LIN {X 0,Y 452.05,Z 502.016,A -85,B 0,C 180,E1 -8755.313,E2 -8755.313} C_VEL
LIN {X 0,Y 450.081,Z 492.867,A -85,B 0,C 180,E1 -8757.12,E2 -8757.12} C_VEL
LIN {X 0,Y 447.199,Z 482.476,A -85,B 0,C 180,E1 -8759.407,E2 -8759.407} C_VEL
LIN {X 0,Y 446.433,Z 480.006,A -85,B 0,C 180,E1 -8760.021,E2 -8760.021} C_VEL
LIN {X 0,Y 446.447,Z 480.002,A -85,B 0,C 180,E1 -8763.454,E2 -8763.454} C_VEL
LIN {X 0,Y 446.404,Z 480.006,A -85,B 0,C 180,E1 -8766.745,E2 -8766.745} C_VEL
LIN {X 0,Y 446.471,Z 479.998,A -85,B 0,C 180,E1 -8769.527,E2 -8769.527} C_VEL
LIN {X 0,Y 446.435,Z 480,A -85,B 0,C 180,E1 -8772.604,E2 -8772.604} C_VEL
LIN {X 0,Y 446.457,Z 480,A -85,B 0,C 180,E1 -8775.103,E2 -8775.103} C_VEL
LIN {X 0,Y 446.431,Z 480.003,A -85,B 0,C 180,E1 -8778.609,E2 -8778.609} C_VEL
LIN {X 0,Y 446.459,Z 480,A -85,B 0,C 180,E1 -8780.974,E2 -8780.974} C_VEL
LIN {X 0,Y 446.423,Z 480.004,A -85,B 0,C 180,E1 -8784.374,E2 -8784.374} C_VEL
LIN {X 0,Y 446.426,Z 480.003,A -85,B 0,C 180,E1 -8787.639,E2 -8787.639} C_VEL
LIN {X 0,Y 446.453,Z 480.14,A -85,B 0,C 180,E1 -8790.791,E2 -8790.791} C_VEL
LIN {X 0,Y 449.137,Z 489.685,A -85,B 0,C 180,E1 -8793.117,E2 -8793.117} C_VEL
LIN {X 0,Y 451.239,Z 500.063,A -85,B 0,C 180,E1 -8795.378,E2 -8795.378} C_VEL
LIN {X 0,Y 451.318,Z 502.583,A -85,B 0,C 180,E1 -8795.872,E2 -8795.872} C_VEL
LIN {X 0,Y 449.674,Z 522.318,A -85,B 0,C 180,E1 -8799.459,E2 -8799.459} C_VEL
LIN {X 0,Y 448.638,Z 537.985,A -85,B 0,C 180,E1 -8802.214,E2 -8802.214} C_VEL
LIN {X 0,Y 448.559,Z 540.298,A -85,B 0,C 180,E1 -8802.575,E2 -8802.575} C_VEL
LIN {X 0,Y 451.577,Z 556.911,A -85,B 0,C 180,E1 -8803.122,E2 -8803.122} C_VEL
LIN {X 0,Y 452.097,Z 561.761,A -85,B 0,C 180,E1 -8803.261,E2 -8803.261} C_VEL
LIN {X 0,Y 450.024,Z 654.195,A -85,B 0,C 180,E1 -8805.183,E2 -8805.183} C_VEL
LIN {X 0,Y 449.587,Z 668.155,A -85,B 0,C 180,E1 -8805.66,E2 -8805.66} C_VEL
LIN {X 0,Y 449.12,Z 681.597,A -85,B 0,C 180,E1 -8806.333,E2 -8806.333} C_VEL
LIN {X 0,Y 448.59,Z 693.288,A -85,B 0,C 180,E1 -8807.1,E2 -8807.1} C_VEL
LIN {X 0,Y 447.989,Z 704.247,A -85,B 0,C 180,E1 -8808.003,E2 -8808.003} C_VEL
LIN {X 0,Y 447.339,Z 715.188,A -85,B 0,C 180,E1 -8809.133,E2 -8809.133} C_VEL
LIN {X 0,Y 446.903,Z 724.107,A -85,B 0,C 180,E1 -8810.267,E2 -8810.267} C_VEL
LIN {X 0,Y 446.363,Z 732.831,A -85,B 0,C 180,E1 -8811.626,E2 -8811.626} C_VEL
LIN {X 0,Y 446.034,Z 740.156,A -85,B 0,C 180,E1 -8813.06,E2 -8813.06} C_VEL
LIN {X 0,Y 445.863,Z 744.583,A -85,B 0,C 180,E1 -8814.119,E2 -8814.119} C_VEL
LIN {X 0,Y 445.641,Z 749.141,A -85,B 0,C 180,E1 -8815.477,E2 -8815.477} C_VEL
LIN {X 0,Y 445.638,Z 751.534,A -85,B 0,C 180,E1 -8816.383,E2 -8816.383} C_VEL
LIN {X 0,Y 445.507,Z 753.496,A -85,B 0,C 180,E1 -8817.287,E2 -8817.287} C_VEL
LIN {X 0,Y 445.412,Z 755.01,A -85,B 0,C 180,E1 -8818.192,E2 -8818.192} C_VEL
LIN {X 0,Y 445.37,Z 756.058,A -85,B 0,C 180,E1 -8819.096,E2 -8819.096} C_VEL
LIN {X 0,Y 445.343,Z 756.704,A -85,B 0,C 180,E1 -8820,E2 -8820} C_VEL
LIN {X 0,Y 445.341,Z 756.949,A -85,B 0,C 180,E1 -8820.904,E2 -8820.904} C_VEL
LIN {X 0,Y 445.379,Z 756.765,A -85,B 0,C 180,E1 -8821.809,E2 -8821.809} C_VEL
LIN {X 0,Y 445.453,Z 756.141,A -85,B 0,C 180,E1 -8822.713,E2 -8822.713} C_VEL
LIN {X 0,Y 445.442,Z 755.119,A -85,B 0,C 180,E1 -8823.618,E2 -8823.618} C_VEL
LIN {X 0,Y 445.439,Z 753.686,A -85,B 0,C 180,E1 -8824.525,E2 -8824.525} C_VEL
LIN {X 0,Y 445.583,Z 750.669,A -85,B 0,C 180,E1 -8825.884,E2 -8825.884} C_VEL
LIN {X 0,Y 445.669,Z 746.583,A -85,B 0,C 180,E1 -8827.248,E2 -8827.248} C_VEL
LIN {X 0,Y 445.945,Z 740.281,A -85,B 0,C 180,E1 -8828.839,E2 -8828.839} C_VEL
LIN {X 0,Y 446.236,Z 733.389,A -85,B 0,C 180,E1 -8830.206,E2 -8830.206} C_VEL
LIN {X 0,Y 446.731,Z 724.835,A -85,B 0,C 180,E1 -8831.571,E2 -8831.571} C_VEL
LIN {X 0,Y 447.063,Z 716.018,A -85,B 0,C 180,E1 -8832.714,E2 -8832.714} C_VEL
LIN {X 0,Y 447.647,Z 705.182,A -85,B 0,C 180,E1 -8833.852,E2 -8833.852} C_VEL
LIN {X 0,Y 448.271,Z 694.465,A -85,B 0,C 180,E1 -8834.76,E2 -8834.76} C_VEL
LIN {X 0,Y 448.76,Z 682.612,A -85,B 0,C 180,E1 -8835.557,E2 -8835.557} C_VEL
LIN {X 0,Y 449.237,Z 669.19,A -85,B 0,C 180,E1 -8836.239,E2 -8836.239} C_VEL
LIN {X 0,Y 449.601,Z 656.633,A -85,B 0,C 180,E1 -8836.692,E2 -8836.692} C_VEL
LIN {X 0,Y 449.911,Z 641.204,A -85,B 0,C 180,E1 -8837.031,E2 -8837.031} C_VEL
LIN {X 0,Y 451.097,Z 559.466,A -85,B 0,C 180,E1 -8838.551,E2 -8838.551} C_VEL
LIN {X 0,Y 448.101,Z 540.66,A -85,B 0,C 180,E1 -8839.052,E2 -8839.052} C_VEL
LIN {X 0,Y 449.102,Z 521.658,A -85,B 0,C 180,E1 -8842.27,E2 -8842.27} C_VEL
LIN {X 0,Y 450.259,Z 502.009,A -85,B 0,C 180,E1 -8845.642,E2 -8845.642} C_VEL
LIN {X 0,Y 450.32,Z 497.645,A -85,B 0,C 180,E1 -8846.41,E2 -8846.41} C_VEL
LIN {X 0,Y 447.487,Z 484.497,A -85,B 0,C 180,E1 -8848.933,E2 -8848.933} C_VEL
LIN {X 0,Y 446.441,Z 480.002,A -85,B 0,C 180,E1 -8849.823,E2 -8849.823} C_VEL
LIN {X 0,Y 446.451,Z 480.001,A -85,B 0,C 180,E1 -8853.433,E2 -8853.433} C_VEL
LIN {X 0,Y 446.411,Z 479.999,A -85,B 0,C 180,E1 -8856.744,E2 -8856.744} C_VEL
LIN {X 0,Y 446.481,Z 479.997,A -85,B 0,C 180,E1 -8859.528,E2 -8859.528} C_VEL
LIN {X 0,Y 446.431,Z 479.996,A -85,B 0,C 180,E1 -8862.604,E2 -8862.604} C_VEL
LIN {X 0,Y 446.454,Z 479.995,A -85,B 0,C 180,E1 -8865.103,E2 -8865.103} C_VEL
LIN {X 0,Y 446.43,Z 479.996,A -85,B 0,C 180,E1 -8868.609,E2 -8868.609} C_VEL
LIN {X 0,Y 446.44,Z 479.996,A -85,B 0,C 180,E1 -8870.972,E2 -8870.972} C_VEL
LIN {X 0,Y 446.421,Z 479.997,A -85,B 0,C 180,E1 -8874.374,E2 -8874.374} C_VEL
LIN {X 0,Y 446.424,Z 480.004,A -85,B 0,C 180,E1 -8877.638,E2 -8877.638} C_VEL
LIN {X 0,Y 446.45,Z 479.994,A -85,B 0,C 180,E1 -8880.791,E2 -8880.791} C_VEL
LIN {X 0,Y 446.461,Z 479.994,A -85,B 0,C 180,E1 -8884.111,E2 -8884.111} C_VEL
LIN {X 0,Y 446.43,Z 479.997,A -85,B 0,C 180,E1 -8886.823,E2 -8886.823} C_VEL
LIN {X 0,Y 446.433,Z 479.998,A -85,B 0,C 180,E1 -8888.036,E2 -8888.036} C_VEL
LIN {X 0,Y 445.804,Z 480.076,A -85,B 0,C 180,E1 -8888.79,E2 -8888.79} C_VEL
LIN {X 0,Y 442.953,Z 480.431,A -85,B 0,C 180,E1 -8890.015,E2 -8890.015} C_VEL
LIN {X 0,Y 440.525,Z 480.734,A -85,B 0,C 180,E1 -8891.003,E2 -8891.003} C_VEL
LIN {X 0,Y 439.495,Z 480.864,A -85,B 0,C 180,E1 -8891.767,E2 -8891.767} C_VEL
LIN {X 0,Y 439.42,Z 480.87,A -85,B 0,C 180,E1 -8892.025,E2 -8892.025} C_VEL
LIN {X 0,Y 439.451,Z 480.869,A -85,B 0,C 180,E1 -8895.174,E2 -8895.174} C_VEL
LIN {X 0,Y 439.486,Z 480.863,A -85,B 0,C 180,E1 -8898.001,E2 -8898.001} C_VEL
LIN {X 0,Y 439.55,Z 480.858,A -85,B 0,C 180,E1 -8901.726,E2 -8901.726} C_VEL
LIN {X 0,Y 439.623,Z 480.844,A -85,B 0,C 180,E1 -8904.496,E2 -8904.496} C_VEL
LIN {X 0,Y 439.637,Z 480.843,A -85,B 0,C 180,E1 -8908.168,E2 -8908.168} C_VEL
LIN {X 0,Y 439.766,Z 480.828,A -85,B 0,C 180,E1 -8910,E2 -8910} C_VEL
LIN {X 0,Y 439.658,Z 480.84,A -85,B 0,C 180,E1 -8912.749,E2 -8912.749} C_VEL
LIN {X 0,Y 439.615,Z 480.845,A -85,B 0,C 180,E1 -8916.425,E2 -8916.425} C_VEL
LIN {X 0,Y 439.501,Z 480.864,A -85,B 0,C 180,E1 -8919.202,E2 -8919.202} C_VEL
LIN {X 0,Y 439.467,Z 480.866,A -85,B 0,C 180,E1 -8922.938,E2 -8922.938} C_VEL
LIN {X 0,Y 439.449,Z 480.866,A -85,B 0,C 180,E1 -8926.349,E2 -8926.349} C_VEL
LIN {X 0,Y 439.404,Z 480.876,A -85,B 0,C 180,E1 -8929.626,E2 -8929.626} C_VEL
LIN {X 0,Y 439.367,Z 480.876,A -85,B 0,C 180,E1 -8932.575,E2 -8932.575} C_VEL
LIN {X 0,Y 439.407,Z 480.876,A -85,B 0,C 180,E1 -8935.585,E2 -8935.585} C_VEL
LIN {X 0,Y 439.419,Z 480.87,A -85,B 0,C 180,E1 -8938.673,E2 -8938.673} C_VEL
LIN {X 0,Y 439.372,Z 480.876,A -85,B 0,C 180,E1 -8942.031,E2 -8942.031} C_VEL
LIN {X 0,Y 439.396,Z 480.881,A -85,B 0,C 180,E1 -8945.34,E2 -8945.34} C_VEL
LIN {X 0,Y 439.386,Z 480.874,A -85,B 0,C 180,E1 -8948.595,E2 -8948.595} C_VEL
LIN {X 0,Y 439.391,Z 480.88,A -85,B 0,C 180,E1 -8951.257,E2 -8951.257} C_VEL
LIN {X 0,Y 439.407,Z 480.872,A -85,B 0,C 180,E1 -8954.729,E2 -8954.729} C_VEL
LIN {X 0,Y 439.397,Z 480.874,A -85,B 0,C 180,E1 -8957.796,E2 -8957.796} C_VEL
LIN {X 0,Y 439.427,Z 480.868,A -85,B 0,C 180,E1 -8960.227,E2 -8960.227} C_VEL
LIN {X 0,Y 439.376,Z 480.878,A -85,B 0,C 180,E1 -8963.713,E2 -8963.713} C_VEL
LIN {X 0,Y 439.375,Z 480.88,A -85,B 0,C 180,E1 -8967.054,E2 -8967.054} C_VEL
LIN {X 0,Y 439.385,Z 480.875,A -85,B 0,C 180,E1 -8970.274,E2 -8970.274} C_VEL
LIN {X 0,Y 439.435,Z 480.978,A -85,B 0,C 180,E1 -8971.598,E2 -8971.598} C_VEL
LIN {X 0,Y 442.64,Z 495.633,A -85,B 0,C 180,E1 -8974.111,E2 -8974.111} C_VEL
LIN {X 0,Y 443.148,Z 500.066,A -85,B 0,C 180,E1 -8974.835,E2 -8974.835} C_VEL
LIN {X 0,Y 442.278,Z 520.819,A -85,B 0,C 180,E1 -8978.073,E2 -8978.073} C_VEL
LIN {X 0,Y 441.486,Z 540.87,A -85,B 0,C 180,E1 -8981.194,E2 -8981.194} C_VEL
LIN {X 0,Y 441.286,Z 546.526,A -85,B 0,C 180,E1 -8982.072,E2 -8982.072} C_VEL
LIN {X 0,Y 443.899,Z 564.854,A -85,B 0,C 180,E1 -8982.535,E2 -8982.535} C_VEL
LIN {X 0,Y 442.597,Z 656.535,A -85,B 0,C 180,E1 -8984.251,E2 -8984.251} C_VEL
LIN {X 0,Y 442.194,Z 670.017,A -85,B 0,C 180,E1 -8984.679,E2 -8984.679} C_VEL
LIN {X 0,Y 441.715,Z 683.289,A -85,B 0,C 180,E1 -8985.311,E2 -8985.311} C_VEL
LIN {X 0,Y 441.247,Z 695.084,A -85,B 0,C 180,E1 -8986.06,E2 -8986.06} C_VEL
LIN {X 0,Y 440.748,Z 706.198,A -85,B 0,C 180,E1 -8986.968,E2 -8986.968} C_VEL
LIN {X 0,Y 440.215,Z 716.607,A -85,B 0,C 180,E1 -8988.022,E2 -8988.022} C_VEL
LIN {X 0,Y 439.718,Z 725.882,A -85,B 0,C 180,E1 -8989.176,E2 -8989.176} C_VEL
LIN {X 0,Y 439.212,Z 734.842,A -85,B 0,C 180,E1 -8990.56,E2 -8990.56} C_VEL
LIN {X 0,Y 438.87,Z 742.06,A -85,B 0,C 180,E1 -8991.945,E2 -8991.945} C_VEL
LIN {X 0,Y 438.645,Z 748.027,A -85,B 0,C 180,E1 -8993.4,E2 -8993.4} C_VEL
LIN {X 0,Y 438.471,Z 752.884,A -85,B 0,C 180,E1 -8994.942,E2 -8994.942} C_VEL
LIN {X 0,Y 438.383,Z 756.075,A -85,B 0,C 180,E1 -8996.323,E2 -8996.323} C_VEL
LIN {X 0,Y 438.389,Z 757.657,A -85,B 0,C 180,E1 -8997.243,E2 -8997.243} C_VEL
LIN {X 0,Y 438.301,Z 758.768,A -85,B 0,C 180,E1 -8998.162,E2 -8998.162} C_VEL
LIN {X 0,Y 438.255,Z 759.464,A -85,B 0,C 180,E1 -8999.081,E2 -8999.081} C_VEL
LIN {X 0,Y 438.253,Z 759.761,A -85,B 0,C 180,E1 -9000,E2 -9000} C_VEL
LIN {X 0,Y 438.255,Z 759.622,A -85,B 0,C 180,E1 -9000.919,E2 -9000.919} C_VEL
LIN {X 0,Y 438.3,Z 759.044,A -85,B 0,C 180,E1 -9001.838,E2 -9001.838} C_VEL
LIN {X 0,Y 438.391,Z 758.064,A -85,B 0,C 180,E1 -9002.757,E2 -9002.757} C_VEL
LIN {X 0,Y 438.404,Z 756.662,A -85,B 0,C 180,E1 -9003.677,E2 -9003.677} C_VEL
LIN {X 0,Y 438.471,Z 753.693,A -85,B 0,C 180,E1 -9005.058,E2 -9005.058} C_VEL
LIN {X 0,Y 438.728,Z 748.75,A -85,B 0,C 180,E1 -9006.693,E2 -9006.693} C_VEL
LIN {X 0,Y 438.971,Z 742.362,A -85,B 0,C 180,E1 -9008.285,E2 -9008.285} C_VEL
LIN {X 0,Y 439.365,Z 735.209,A -85,B 0,C 180,E1 -9009.669,E2 -9009.669} C_VEL
LIN {X 0,Y 439.835,Z 726.323,A -85,B 0,C 180,E1 -9011.055,E2 -9011.055} C_VEL
LIN {X 0,Y 440.485,Z 716.065,A -85,B 0,C 180,E1 -9012.322,E2 -9012.322} C_VEL
LIN {X 0,Y 441.026,Z 705.55,A -85,B 0,C 180,E1 -9013.371,E2 -9013.371} C_VEL
LIN {X 0,Y 441.563,Z 694.039,A -85,B 0,C 180,E1 -9014.282,E2 -9014.282} C_VEL
LIN {X 0,Y 442.067,Z 682.933,A -85,B 0,C 180,E1 -9014.972,E2 -9014.972} C_VEL
LIN {X 0,Y 442.533,Z 670.892,A -85,B 0,C 180,E1 -9015.545,E2 -9015.545} C_VEL
LIN {X 0,Y 442.905,Z 657.826,A -85,B 0,C 180,E1 -9015.975,E2 -9015.975} C_VEL
LIN {X 0,Y 444.641,Z 563.555,A -85,B 0,C 180,E1 -9017.869,E2 -9017.869} C_VEL
LIN {X 0,Y 441.922,Z 547.719,A -85,B 0,C 180,E1 -9018.368,E2 -9018.368} C_VEL
LIN {X 0,Y 442.726,Z 526.147,A -85,B 0,C 180,E1 -9021.659,E2 -9021.659} C_VEL
LIN {X 0,Y 443.633,Z 505.304,A -85,B 0,C 180,E1 -9024.823,E2 -9024.823} C_VEL
LIN {X 0,Y 443.662,Z 498.749,A -85,B 0,C 180,E1 -9025.825,E2 -9025.825} C_VEL
LIN {X 0,Y 441.267,Z 487.476,A -85,B 0,C 180,E1 -9027.744,E2 -9027.744} C_VEL
LIN {X 0,Y 439.446,Z 480.874,A -85,B 0,C 180,E1 -9028.933,E2 -9028.933} C_VEL
LIN {X 0,Y 439.373,Z 480.884,A -85,B 0,C 180,E1 -9032.03,E2 -9032.03} C_VEL
LIN {X 0,Y 439.397,Z 480.878,A -85,B 0,C 180,E1 -9035.34,E2 -9035.34} C_VEL
LIN {X 0,Y 439.385,Z 480.879,A -85,B 0,C 180,E1 -9038.595,E2 -9038.595} C_VEL
LIN {X 0,Y 439.39,Z 480.877,A -85,B 0,C 180,E1 -9041.257,E2 -9041.257} C_VEL
LIN {X 0,Y 439.404,Z 480.877,A -85,B 0,C 180,E1 -9044.729,E2 -9044.729} C_VEL
LIN {X 0,Y 439.4,Z 480.875,A -85,B 0,C 180,E1 -9047.796,E2 -9047.796} C_VEL
LIN {X 0,Y 439.439,Z 480.874,A -85,B 0,C 180,E1 -9050.228,E2 -9050.228} C_VEL
LIN {X 0,Y 439.379,Z 480.878,A -85,B 0,C 180,E1 -9053.713,E2 -9053.713} C_VEL
LIN {X 0,Y 439.377,Z 480.879,A -85,B 0,C 180,E1 -9057.054,E2 -9057.054} C_VEL
LIN {X 0,Y 439.438,Z 480.874,A -85,B 0,C 180,E1 -9060.804,E2 -9060.804} C_VEL
LIN {X 0,Y 439.474,Z 480.999,A -85,B 0,C 180,E1 -9061.233,E2 -9061.233} C_VEL
LIN {X 0,Y 443.439,Z 497.52,A -85,B 0,C 180,E1 -9064.149,E2 -9064.149} C_VEL
LIN {X 0,Y 444.397,Z 502.382,A -85,B 0,C 180,E1 -9064.973,E2 -9064.973} C_VEL
LIN {X 0,Y 442.89,Z 524.545,A -85,B 0,C 180,E1 -9068.35,E2 -9068.35} C_VEL
LIN {X 0,Y 442.849,Z 525.695,A -85,B 0,C 180,E1 -9068.485,E2 -9068.485} C_VEL
LIN {X 0,Y 445.968,Z 545.988,A -85,B 0,C 180,E1 -9069.007,E2 -9069.007} C_VEL
LIN {X 0,Y 444.046,Z 662.624,A -85,B 0,C 180,E1 -9071.127,E2 -9071.127} C_VEL
LIN {X 0,Y 443.555,Z 677.086,A -85,B 0,C 180,E1 -9071.575,E2 -9071.575} C_VEL
LIN {X 0,Y 443.021,Z 691.131,A -85,B 0,C 180,E1 -9072.204,E2 -9072.204} C_VEL
LIN {X 0,Y 442.484,Z 703.157,A -85,B 0,C 180,E1 -9072.912,E2 -9072.912} C_VEL
LIN {X 0,Y 441.698,Z 715.682,A -85,B 0,C 180,E1 -9073.832,E2 -9073.832} C_VEL
LIN {X 0,Y 441.014,Z 727.136,A -85,B 0,C 180,E1 -9074.873,E2 -9074.873} C_VEL
LIN {X 0,Y 440.246,Z 738.604,A -85,B 0,C 180,E1 -9076.145,E2 -9076.145} C_VEL
LIN {X 0,Y 439.747,Z 748.996,A -85,B 0,C 180,E1 -9077.566,E2 -9077.566} C_VEL
LIN {X 0,Y 439.237,Z 757.274,A -85,B 0,C 180,E1 -9078.93,E2 -9078.93} C_VEL
LIN {X 0,Y 438.83,Z 765.321,A -85,B 0,C 180,E1 -9080.552,E2 -9080.552} C_VEL
LIN {X 0,Y 438.529,Z 771.754,A -85,B 0,C 180,E1 -9082.171,E2 -9082.171} C_VEL
LIN {X 0,Y 438.442,Z 776.349,A -85,B 0,C 180,E1 -9083.631,E2 -9083.631} C_VEL
LIN {X 0,Y 438.321,Z 780.535,A -85,B 0,C 180,E1 -9085.402,E2 -9085.402} C_VEL
LIN {X 0,Y 438.337,Z 783.411,A -85,B 0,C 180,E1 -9087.243,E2 -9087.243} C_VEL
LIN {X 0,Y 438.252,Z 784.843,A -85,B 0,C 180,E1 -9089.081,E2 -9089.081} C_VEL
LIN {X 0,Y 438.252,Z 784.854,A -85,B 0,C 180,E1 -9090.919,E2 -9090.919} C_VEL
LIN {X 0,Y 438.337,Z 783.426,A -85,B 0,C 180,E1 -9092.757,E2 -9092.757} C_VEL
LIN {X 0,Y 438.321,Z 780.547,A -85,B 0,C 180,E1 -9094.598,E2 -9094.598} C_VEL
LIN {X 0,Y 438.447,Z 776.153,A -85,B 0,C 180,E1 -9096.443,E2 -9096.443} C_VEL
LIN {X 0,Y 438.525,Z 771.78,A -85,B 0,C 180,E1 -9097.83,E2 -9097.83} C_VEL
LIN {X 0,Y 438.818,Z 765.357,A -85,B 0,C 180,E1 -9099.449,E2 -9099.449} C_VEL
LIN {X 0,Y 439.232,Z 757.324,A -85,B 0,C 180,E1 -9101.07,E2 -9101.07} C_VEL
LIN {X 0,Y 439.779,Z 748.08,A -85,B 0,C 180,E1 -9102.587,E2 -9102.587} C_VEL
LIN {X 0,Y 440.295,Z 738.736,A -85,B 0,C 180,E1 -9103.853,E2 -9103.853} C_VEL
LIN {X 0,Y 440.979,Z 727.39,A -85,B 0,C 180,E1 -9105.128,E2 -9105.128} C_VEL
LIN {X 0,Y 441.687,Z 716.073,A -85,B 0,C 180,E1 -9106.168,E2 -9106.168} C_VEL
LIN {X 0,Y 442.483,Z 703.72,A -85,B 0,C 180,E1 -9107.088,E2 -9107.088} C_VEL
LIN {X 0,Y 443.135,Z 690.483,A -85,B 0,C 180,E1 -9107.87,E2 -9107.87} C_VEL
LIN {X 0,Y 443.743,Z 675.682,A -85,B 0,C 180,E1 -9108.527,E2 -9108.527} C_VEL
LIN {X 0,Y 444.265,Z 661.645,A -85,B 0,C 180,E1 -9108.953,E2 -9108.953} C_VEL
LIN {X 0,Y 446.318,Z 552.911,A -85,B 0,C 180,E1 -9111.032,E2 -9111.032} C_VEL
LIN {X 0,Y 446.402,Z 545.094,A -85,B 0,C 180,E1 -9111.194,E2 -9111.194} C_VEL
LIN {X 0,Y 444.191,Z 530.718,A -85,B 0,C 180,E1 -9111.634,E2 -9111.634} C_VEL
LIN {X 0,Y 443.391,Z 526.521,A -85,B 0,C 180,E1 -9111.793,E2 -9111.793} C_VEL
LIN {X 0,Y 445.31,Z 507.027,A -85,B 0,C 180,E1 -9114.972,E2 -9114.972} C_VEL
LIN {X 0,Y 445.319,Z 503.632,A -85,B 0,C 180,E1 -9115.58,E2 -9115.58} C_VEL
LIN {X 0,Y 443.118,Z 493.62,A -85,B 0,C 180,E1 -9117.64,E2 -9117.64} C_VEL
LIN {X 0,Y 439.987,Z 482.961,A -85,B 0,C 180,E1 -9120.132,E2 -9120.132} C_VEL
LIN {X 0,Y 439.362,Z 480.886,A -85,B 0,C 180,E1 -9120.712,E2 -9120.712} C_VEL
LIN {X 0,Y 439.389,Z 480.88,A -85,B 0,C 180,E1 -9124.044,E2 -9124.044} C_VEL
LIN {X 0,Y 439.35,Z 480.884,A -85,B 0,C 180,E1 -9126.887,E2 -9126.887} C_VEL
LIN {X 0,Y 439.409,Z 480.876,A -85,B 0,C 180,E1 -9129.85,E2 -9129.85} C_VEL
LIN {X 0,Y 439.388,Z 480.878,A -85,B 0,C 180,E1 -9132.628,E2 -9132.628} C_VEL
LIN {X 0,Y 439.405,Z 480.877,A -85,B 0,C 180,E1 -9135.271,E2 -9135.271} C_VEL
LIN {X 0,Y 439.391,Z 480.88,A -85,B 0,C 180,E1 -9138.743,E2 -9138.743} C_VEL
LIN {X 0,Y 439.379,Z 480.881,A -85,B 0,C 180,E1 -9141.607,E2 -9141.607} C_VEL
LIN {X 0,Y 439.402,Z 480.88,A -85,B 0,C 180,E1 -9144.844,E2 -9144.844} C_VEL
LIN {X 0,Y 439.377,Z 480.881,A -85,B 0,C 180,E1 -9148.14,E2 -9148.14} C_VEL
LIN {X 0,Y 439.401,Z 480.972,A -85,B 0,C 180,E1 -9150.137,E2 -9150.137} C_VEL
LIN {X 0,Y 442.403,Z 491.514,A -85,B 0,C 180,E1 -9152.825,E2 -9152.825} C_VEL
LIN {X 0,Y 444.372,Z 500.982,A -85,B 0,C 180,E1 -9154.972,E2 -9154.972} C_VEL
LIN {X 0,Y 444.725,Z 503.411,A -85,B 0,C 180,E1 -9155.491,E2 -9155.491} C_VEL
LIN {X 0,Y 442.962,Z 523.022,A -85,B 0,C 180,E1 -9159.134,E2 -9159.134} C_VEL
LIN {X 0,Y 441.785,Z 539.267,A -85,B 0,C 180,E1 -9162.052,E2 -9162.052} C_VEL
LIN {X 0,Y 441.805,Z 540.203,A -85,B 0,C 180,E1 -9162.169,E2 -9162.169} C_VEL
LIN {X 0,Y 444.963,Z 557.327,A -85,B 0,C 180,E1 -9162.771,E2 -9162.771} C_VEL
LIN {X 0,Y 445.523,Z 562.72,A -85,B 0,C 180,E1 -9162.932,E2 -9162.932} C_VEL
LIN {X 0,Y 443.28,Z 654.232,A -85,B 0,C 180,E1 -9164.894,E2 -9164.894} C_VEL
LIN {X 0,Y 442.83,Z 668.089,A -85,B 0,C 180,E1 -9165.38,E2 -9165.38} C_VEL
LIN {X 0,Y 442.356,Z 681.069,A -85,B 0,C 180,E1 -9166.037,E2 -9166.037} C_VEL
LIN {X 0,Y 441.706,Z 693.958,A -85,B 0,C 180,E1 -9166.895,E2 -9166.895} C_VEL
LIN {X 0,Y 441.074,Z 704.807,A -85,B 0,C 180,E1 -9167.812,E2 -9167.812} C_VEL
LIN {X 0,Y 440.396,Z 715.704,A -85,B 0,C 180,E1 -9168.96,E2 -9168.96} C_VEL
LIN {X 0,Y 439.932,Z 724.592,A -85,B 0,C 180,E1 -9170.111,E2 -9170.111} C_VEL
LIN {X 0,Y 439.355,Z 733.264,A -85,B 0,C 180,E1 -9171.491,E2 -9171.491} C_VEL
LIN {X 0,Y 438.987,Z 740.884,A -85,B 0,C 180,E1 -9173.026,E2 -9173.026} C_VEL
LIN {X 0,Y 438.83,Z 744.93,A -85,B 0,C 180,E1 -9174.025,E2 -9174.025} C_VEL
LIN {X 0,Y 438.557,Z 749.459,A -85,B 0,C 180,E1 -9175.404,E2 -9175.404} C_VEL
LIN {X 0,Y 438.582,Z 751.844,A -85,B 0,C 180,E1 -9176.325,E2 -9176.325} C_VEL
LIN {X 0,Y 438.438,Z 753.797,A -85,B 0,C 180,E1 -9177.244,E2 -9177.244} C_VEL
LIN {X 0,Y 438.332,Z 755.289,A -85,B 0,C 180,E1 -9178.162,E2 -9178.162} C_VEL
LIN {X 0,Y 438.282,Z 756.326,A -85,B 0,C 180,E1 -9179.081,E2 -9179.081} C_VEL
LIN {X 0,Y 438.254,Z 756.958,A -85,B 0,C 180,E1 -9180,E2 -9180} C_VEL
LIN {X 0,Y 438.255,Z 757.187,A -85,B 0,C 180,E1 -9180.919,E2 -9180.919} C_VEL
LIN {X 0,Y 438.3,Z 756.97,A -85,B 0,C 180,E1 -9181.838,E2 -9181.838} C_VEL
LIN {X 0,Y 438.38,Z 756.327,A -85,B 0,C 180,E1 -9182.757,E2 -9182.757} C_VEL
LIN {X 0,Y 438.344,Z 755.28,A -85,B 0,C 180,E1 -9183.677,E2 -9183.677} C_VEL
LIN {X 0,Y 438.365,Z 753.819,A -85,B 0,C 180,E1 -9184.598,E2 -9184.598} C_VEL
LIN {X 0,Y 438.487,Z 750.335,A -85,B 0,C 180,E1 -9186.136,E2 -9186.136} C_VEL
LIN {X 0,Y 438.681,Z 744.948,A -85,B 0,C 180,E1 -9187.827,E2 -9187.827} C_VEL
LIN {X 0,Y 438.937,Z 739.175,A -85,B 0,C 180,E1 -9189.213,E2 -9189.213} C_VEL
LIN {X 0,Y 439.254,Z 731.96,A -85,B 0,C 180,E1 -9190.603,E2 -9190.603} C_VEL
LIN {X 0,Y 439.824,Z 722.925,A -85,B 0,C 180,E1 -9191.989,E2 -9191.989} C_VEL
LIN {X 0,Y 440.223,Z 713.82,A -85,B 0,C 180,E1 -9193.132,E2 -9193.132} C_VEL
LIN {X 0,Y 440.811,Z 703.502,A -85,B 0,C 180,E1 -9194.189,E2 -9194.189} C_VEL
LIN {X 0,Y 441.458,Z 692.254,A -85,B 0,C 180,E1 -9195.111,E2 -9195.111} C_VEL
LIN {X 0,Y 441.966,Z 679.765,A -85,B 0,C 180,E1 -9195.921,E2 -9195.921} C_VEL
LIN {X 0,Y 442.355,Z 668.048,A -85,B 0,C 180,E1 -9196.499,E2 -9196.499} C_VEL
LIN {X 0,Y 442.822,Z 654.749,A -85,B 0,C 180,E1 -9196.955,E2 -9196.955} C_VEL
LIN {X 0,Y 443.146,Z 636.912,A -85,B 0,C 180,E1 -9197.329,E2 -9197.329} C_VEL
LIN {X 0,Y 444.371,Z 560.785,A -85,B 0,C 180,E1 -9198.784,E2 -9198.784} C_VEL
LIN {X 0,Y 441.168,Z 540.605,A -85,B 0,C 180,E1 -9199.333,E2 -9199.333} C_VEL
LIN {X 0,Y 442.387,Z 519.198,A -85,B 0,C 180,E1 -9203.011,E2 -9203.011} C_VEL
LIN {X 0,Y 443.532,Z 500.154,A -85,B 0,C 180,E1 -9206.339,E2 -9206.339} C_VEL
LIN {X 0,Y 441.231,Z 488.712,A -85,B 0,C 180,E1 -9208.545,E2 -9208.545} C_VEL
LIN {X 0,Y 439.403,Z 480.878,A -85,B 0,C 180,E1 -9210.134,E2 -9210.134} C_VEL
LIN {X 0,Y 439.399,Z 480.879,A -85,B 0,C 180,E1 -9213.724,E2 -9213.724} C_VEL
LIN {X 0,Y 439.359,Z 480.878,A -85,B 0,C 180,E1 -9216.888,E2 -9216.888} C_VEL
LIN {X 0,Y 439.415,Z 480.875,A -85,B 0,C 180,E1 -9219.851,E2 -9219.851} C_VEL
LIN {X 0,Y 439.384,Z 480.874,A -85,B 0,C 180,E1 -9222.627,E2 -9222.627} C_VEL
LIN {X 0,Y 439.402,Z 480.876,A -85,B 0,C 180,E1 -9225.27,E2 -9225.27} C_VEL
LIN {X 0,Y 439.39,Z 480.873,A -85,B 0,C 180,E1 -9228.743,E2 -9228.743} C_VEL
LIN {X 0,Y 439.374,Z 480.883,A -85,B 0,C 180,E1 -9231.608,E2 -9231.608} C_VEL
LIN {X 0,Y 439.401,Z 480.872,A -85,B 0,C 180,E1 -9234.844,E2 -9234.844} C_VEL
LIN {X 0,Y 439.375,Z 480.876,A -85,B 0,C 180,E1 -9238.139,E2 -9238.139} C_VEL
LIN {X 0,Y 439.434,Z 480.875,A -85,B 0,C 180,E1 -9241.598,E2 -9241.598} C_VEL
LIN {X 0,Y 439.407,Z 480.871,A -85,B 0,C 180,E1 -9244.415,E2 -9244.415} C_VEL
LIN {X 0,Y 439.367,Z 480.883,A -85,B 0,C 180,E1 -9247.424,E2 -9247.424} C_VEL
LIN {X 0,Y 439.443,Z 480.867,A -85,B 0,C 180,E1 -9250.663,E2 -9250.663} C_VEL
LIN {X 0,Y 439.42,Z 480.87,A -85,B 0,C 180,E1 -9252.025,E2 -9252.025} C_VEL
LIN {X 0,Y 438.775,Z 480.951,A -85,B 0,C 180,E1 -9252.79,E2 -9252.79} C_VEL
LIN {X 0,Y 435.926,Z 481.309,A -85,B 0,C 180,E1 -9254.033,E2 -9254.033} C_VEL
LIN {X 0,Y 433.501,Z 481.612,A -85,B 0,C 180,E1 -9255.036,E2 -9255.036} C_VEL
LIN {X 0,Y 432.459,Z 481.741,A -85,B 0,C 180,E1 -9255.811,E2 -9255.811} C_VEL
LIN {X 0,Y 432.374,Z 481.749,A -85,B 0,C 180,E1 -9256.073,E2 -9256.073} C_VEL
LIN {X 0,Y 432.395,Z 481.745,A -85,B 0,C 180,E1 -9258.753,E2 -9258.753} C_VEL
LIN {X 0,Y 432.588,Z 481.721,A -85,B 0,C 180,E1 -9262.321,E2 -9262.321} C_VEL
LIN {X 0,Y 432.6,Z 481.719,A -85,B 0,C 180,E1 -9264.406,E2 -9264.406} C_VEL
LIN {X 0,Y 432.607,Z 481.719,A -85,B 0,C 180,E1 -9268.138,E2 -9268.138} C_VEL
LIN {X 0,Y 432.736,Z 481.704,A -85,B 0,C 180,E1 -9270,E2 -9270} C_VEL
LIN {X 0,Y 432.608,Z 481.719,A -85,B 0,C 180,E1 -9272.793,E2 -9272.793} C_VEL
LIN {X 0,Y 432.571,Z 481.723,A -85,B 0,C 180,E1 -9276.53,E2 -9276.53} C_VEL
LIN {X 0,Y 432.444,Z 481.745,A -85,B 0,C 180,E1 -9279.353,E2 -9279.353} C_VEL
LIN {X 0,Y 432.432,Z 481.741,A -85,B 0,C 180,E1 -9282.804,E2 -9282.804} C_VEL
LIN {X 0,Y 432.414,Z 481.742,A -85,B 0,C 180,E1 -9286.479,E2 -9286.479} C_VEL
LIN {X 0,Y 432.34,Z 481.753,A -85,B 0,C 180,E1 -9289.96,E2 -9289.96} C_VEL
LIN {X 0,Y 432.322,Z 481.756,A -85,B 0,C 180,E1 -9292.964,E2 -9292.964} C_VEL
LIN {X 0,Y 432.366,Z 481.749,A -85,B 0,C 180,E1 -9296.032,E2 -9296.032} C_VEL
LIN {X 0,Y 432.345,Z 481.756,A -85,B 0,C 180,E1 -9299.187,E2 -9299.187} C_VEL
LIN {X 0,Y 432.324,Z 481.753,A -85,B 0,C 180,E1 -9302.443,E2 -9302.443} C_VEL
LIN {X 0,Y 432.345,Z 481.755,A -85,B 0,C 180,E1 -9305.632,E2 -9305.632} C_VEL
LIN {X 0,Y 432.356,Z 481.757,A -85,B 0,C 180,E1 -9309.342,E2 -9309.342} C_VEL
LIN {X 0,Y 432.337,Z 481.754,A -85,B 0,C 180,E1 -9311.797,E2 -9311.797} C_VEL
LIN {X 0,Y 432.342,Z 481.751,A -85,B 0,C 180,E1 -9314.346,E2 -9314.346} C_VEL
LIN {X 0,Y 432.322,Z 481.758,A -85,B 0,C 180,E1 -9317.016,E2 -9317.016} C_VEL
LIN {X 0,Y 432.335,Z 481.754,A -85,B 0,C 180,E1 -9319.821,E2 -9319.821} C_VEL
LIN {X 0,Y 432.308,Z 481.76,A -85,B 0,C 180,E1 -9323.022,E2 -9323.022} C_VEL
LIN {X 0,Y 432.361,Z 481.75,A -85,B 0,C 180,E1 -9325.997,E2 -9325.997} C_VEL
LIN {X 0,Y 432.35,Z 481.755,A -85,B 0,C 180,E1 -9329.49,E2 -9329.49} C_VEL
LIN {X 0,Y 432.404,Z 481.912,A -85,B 0,C 180,E1 -9331.364,E2 -9331.364} C_VEL
LIN {X 0,Y 435.667,Z 496.741,A -85,B 0,C 180,E1 -9333.923,E2 -9333.923} C_VEL
LIN {X 0,Y 436.264,Z 500.883,A -85,B 0,C 180,E1 -9334.618,E2 -9334.618} C_VEL
LIN {X 0,Y 435.44,Z 520.507,A -85,B 0,C 180,E1 -9337.71,E2 -9337.71} C_VEL
LIN {X 0,Y 434.659,Z 539.198,A -85,B 0,C 180,E1 -9340.642,E2 -9340.642} C_VEL
LIN {X 0,Y 434.404,Z 547,A -85,B 0,C 180,E1 -9341.828,E2 -9341.828} C_VEL
LIN {X 0,Y 437.067,Z 564.816,A -85,B 0,C 180,E1 -9342.285,E2 -9342.285} C_VEL
LIN {X 0,Y 435.674,Z 657.022,A -85,B 0,C 180,E1 -9344.054,E2 -9344.054} C_VEL
LIN {X 0,Y 435.274,Z 670.352,A -85,B 0,C 180,E1 -9344.489,E2 -9344.489} C_VEL
LIN {X 0,Y 434.773,Z 683.57,A -85,B 0,C 180,E1 -9345.131,E2 -9345.131} C_VEL
LIN {X 0,Y 434.231,Z 696.1,A -85,B 0,C 180,E1 -9345.95,E2 -9345.95} C_VEL
LIN {X 0,Y 433.714,Z 707.236,A -85,B 0,C 180,E1 -9346.888,E2 -9346.888} C_VEL
LIN {X 0,Y 433.17,Z 717.373,A -85,B 0,C 180,E1 -9347.943,E2 -9347.943} C_VEL
LIN {X 0,Y 432.688,Z 725.706,A -85,B 0,C 180,E1 -9348.998,E2 -9348.998} C_VEL
LIN {X 0,Y 432.188,Z 734.746,A -85,B 0,C 180,E1 -9350.405,E2 -9350.405} C_VEL
LIN {X 0,Y 431.806,Z 742.027,A -85,B 0,C 180,E1 -9351.812,E2 -9351.812} C_VEL
LIN {X 0,Y 431.564,Z 748.467,A -85,B 0,C 180,E1 -9353.407,E2 -9353.407} C_VEL
LIN {X 0,Y 431.41,Z 752.968,A -85,B 0,C 180,E1 -9354.859,E2 -9354.859} C_VEL
LIN {X 0,Y 431.286,Z 756.198,A -85,B 0,C 180,E1 -9356.263,E2 -9356.263} C_VEL
LIN {X 0,Y 431.301,Z 757.798,A -85,B 0,C 180,E1 -9357.198,E2 -9357.198} C_VEL
LIN {X 0,Y 431.225,Z 758.934,A -85,B 0,C 180,E1 -9358.132,E2 -9358.132} C_VEL
LIN {X 0,Y 431.172,Z 759.645,A -85,B 0,C 180,E1 -9359.066,E2 -9359.066} C_VEL
LIN {X 0,Y 431.167,Z 759.953,A -85,B 0,C 180,E1 -9360,E2 -9360} C_VEL
LIN {X 0,Y 431.172,Z 759.834,A -85,B 0,C 180,E1 -9360.934,E2 -9360.934} C_VEL
LIN {X 0,Y 431.225,Z 759.266,A -85,B 0,C 180,E1 -9361.868,E2 -9361.868} C_VEL
LIN {X 0,Y 431.321,Z 758.296,A -85,B 0,C 180,E1 -9362.802,E2 -9362.802} C_VEL
LIN {X 0,Y 431.311,Z 756.912,A -85,B 0,C 180,E1 -9363.737,E2 -9363.737} C_VEL
LIN {X 0,Y 431.417,Z 753.965,A -85,B 0,C 180,E1 -9365.14,E2 -9365.14} C_VEL
LIN {X 0,Y 431.665,Z 749.369,A -85,B 0,C 180,E1 -9366.708,E2 -9366.708} C_VEL
LIN {X 0,Y 431.895,Z 743.678,A -85,B 0,C 180,E1 -9368.186,E2 -9368.186} C_VEL
LIN {X 0,Y 432.325,Z 736.833,A -85,B 0,C 180,E1 -9369.592,E2 -9369.592} C_VEL
LIN {X 0,Y 432.807,Z 728.227,A -85,B 0,C 180,E1 -9370.999,E2 -9370.999} C_VEL
LIN {X 0,Y 433.355,Z 719.396,A -85,B 0,C 180,E1 -9372.171,E2 -9372.171} C_VEL
LIN {X 0,Y 433.935,Z 709.731,A -85,B 0,C 180,E1 -9373.227,E2 -9373.227} C_VEL
LIN {X 0,Y 434.492,Z 699.164,A -85,B 0,C 180,E1 -9374.161,E2 -9374.161} C_VEL
LIN {X 0,Y 434.965,Z 687.537,A -85,B 0,C 180,E1 -9374.982,E2 -9374.982} C_VEL
LIN {X 0,Y 435.572,Z 675.684,A -85,B 0,C 180,E1 -9375.62,E2 -9375.62} C_VEL
LIN {X 0,Y 436.034,Z 661.995,A -85,B 0,C 180,E1 -9376.143,E2 -9376.143} C_VEL
LIN {X 0,Y 436.315,Z 648.758,A -85,B 0,C 180,E1 -9376.463,E2 -9376.463} C_VEL
LIN {X 0,Y 437.97,Z 567.728,A -85,B 0,C 180,E1 -9378.127,E2 -9378.127} C_VEL
LIN {X 0,Y 437.841,Z 563.434,A -85,B 0,C 180,E1 -9378.232,E2 -9378.232} C_VEL
LIN {X 0,Y 435.19,Z 547.922,A -85,B 0,C 180,E1 -9378.746,E2 -9378.746} C_VEL
LIN {X 0,Y 436.127,Z 525.243,A -85,B 0,C 180,E1 -9382.253,E2 -9382.253} C_VEL
LIN {X 0,Y 437.056,Z 504.817,A -85,B 0,C 180,E1 -9385.385,E2 -9385.385} C_VEL
LIN {X 0,Y 437.011,Z 500.908,A -85,B 0,C 180,E1 -9385.991,E2 -9385.991} C_VEL
LIN {X 0,Y 435.014,Z 491.144,A -85,B 0,C 180,E1 -9387.687,E2 -9387.687} C_VEL
LIN {X 0,Y 432.364,Z 481.755,A -85,B 0,C 180,E1 -9389.42,E2 -9389.42} C_VEL
LIN {X 0,Y 432.325,Z 481.762,A -85,B 0,C 180,E1 -9392.443,E2 -9392.443} C_VEL
LIN {X 0,Y 432.346,Z 481.755,A -85,B 0,C 180,E1 -9395.632,E2 -9395.632} C_VEL
LIN {X 0,Y 432.352,Z 481.754,A -85,B 0,C 180,E1 -9399.343,E2 -9399.343} C_VEL
LIN {X 0,Y 432.335,Z 481.755,A -85,B 0,C 180,E1 -9401.797,E2 -9401.797} C_VEL
LIN {X 0,Y 432.335,Z 481.757,A -85,B 0,C 180,E1 -9404.347,E2 -9404.347} C_VEL
LIN {X 0,Y 432.327,Z 481.756,A -85,B 0,C 180,E1 -9407.015,E2 -9407.015} C_VEL
LIN {X 0,Y 432.343,Z 481.755,A -85,B 0,C 180,E1 -9409.819,E2 -9409.819} C_VEL
LIN {X 0,Y 432.317,Z 481.759,A -85,B 0,C 180,E1 -9413.023,E2 -9413.023} C_VEL
LIN {X 0,Y 432.361,Z 481.753,A -85,B 0,C 180,E1 -9415.996,E2 -9415.996} C_VEL
LIN {X 0,Y 432.397,Z 481.751,A -85,B 0,C 180,E1 -9419.744,E2 -9419.744} C_VEL
LIN {X 0,Y 432.431,Z 481.946,A -85,B 0,C 180,E1 -9420.931,E2 -9420.931} C_VEL
LIN {X 0,Y 436.15,Z 497.326,A -85,B 0,C 180,E1 -9423.696,E2 -9423.696} C_VEL
LIN {X 0,Y 437.494,Z 503.718,A -85,B 0,C 180,E1 -9424.805,E2 -9424.805} C_VEL
LIN {X 0,Y 436.159,Z 522.728,A -85,B 0,C 180,E1 -9427.749,E2 -9427.749} C_VEL
LIN {X 0,Y 435.996,Z 525.507,A -85,B 0,C 180,E1 -9428.176,E2 -9428.176} C_VEL
LIN {X 0,Y 439.21,Z 546.401,A -85,B 0,C 180,E1 -9428.731,E2 -9428.731} C_VEL
LIN {X 0,Y 437.217,Z 662.067,A -85,B 0,C 180,E1 -9430.882,E2 -9430.882} C_VEL
LIN {X 0,Y 436.709,Z 676.737,A -85,B 0,C 180,E1 -9431.34,E2 -9431.34} C_VEL
LIN {X 0,Y 436.096,Z 691.42,A -85,B 0,C 180,E1 -9432.009,E2 -9432.009} C_VEL
LIN {X 0,Y 435.534,Z 703.709,A -85,B 0,C 180,E1 -9432.752,E2 -9432.752} C_VEL
LIN {X 0,Y 434.712,Z 716.101,A -85,B 0,C 180,E1 -9433.686,E2 -9433.686} C_VEL
LIN {X 0,Y 434.011,Z 727.468,A -85,B 0,C 180,E1 -9434.744,E2 -9434.744} C_VEL
LIN {X 0,Y 433.282,Z 737.906,A -85,B 0,C 180,E1 -9435.918,E2 -9435.918} C_VEL
LIN {X 0,Y 432.777,Z 747.04,A -85,B 0,C 180,E1 -9437.153,E2 -9437.153} C_VEL
LIN {X 0,Y 432.221,Z 756.771,A -85,B 0,C 180,E1 -9438.748,E2 -9438.748} C_VEL
LIN {X 0,Y 431.782,Z 764.885,A -85,B 0,C 180,E1 -9440.396,E2 -9440.396} C_VEL
LIN {X 0,Y 431.47,Z 771.374,A -85,B 0,C 180,E1 -9442.042,E2 -9442.042} C_VEL
LIN {X 0,Y 431.336,Z 776.412,A -85,B 0,C 180,E1 -9443.673,E2 -9443.673} C_VEL
LIN {X 0,Y 431.247,Z 780.24,A -85,B 0,C 180,E1 -9445.326,E2 -9445.326} C_VEL
LIN {X 0,Y 431.232,Z 783.145,A -85,B 0,C 180,E1 -9447.198,E2 -9447.198} C_VEL
LIN {X 0,Y 431.169,Z 784.6,A -85,B 0,C 180,E1 -9449.066,E2 -9449.066} C_VEL
LIN {X 0,Y 431.169,Z 784.631,A -85,B 0,C 180,E1 -9450.934,E2 -9450.934} C_VEL
LIN {X 0,Y 431.232,Z 783.216,A -85,B 0,C 180,E1 -9452.803,E2 -9452.803} C_VEL
LIN {X 0,Y 431.248,Z 780.341,A -85,B 0,C 180,E1 -9454.674,E2 -9454.674} C_VEL
LIN {X 0,Y 431.372,Z 775.941,A -85,B 0,C 180,E1 -9456.549,E2 -9456.549} C_VEL
LIN {X 0,Y 431.548,Z 769.895,A -85,B 0,C 180,E1 -9458.428,E2 -9458.428} C_VEL
LIN {X 0,Y 431.851,Z 763.057,A -85,B 0,C 180,E1 -9460.076,E2 -9460.076} C_VEL
LIN {X 0,Y 432.39,Z 754.488,A -85,B 0,C 180,E1 -9461.723,E2 -9461.723} C_VEL
LIN {X 0,Y 432.921,Z 745.525,A -85,B 0,C 180,E1 -9463.137,E2 -9463.137} C_VEL
LIN {X 0,Y 433.579,Z 734.628,A -85,B 0,C 180,E1 -9464.551,E2 -9464.551} C_VEL
LIN {X 0,Y 434.312,Z 723.598,A -85,B 0,C 180,E1 -9465.727,E2 -9465.727} C_VEL
LIN {X 0,Y 435.124,Z 711.538,A -85,B 0,C 180,E1 -9466.781,E2 -9466.781} C_VEL
LIN {X 0,Y 435.965,Z 698.133,A -85,B 0,C 180,E1 -9467.715,E2 -9467.715} C_VEL
LIN {X 0,Y 436.634,Z 685.231,A -85,B 0,C 180,E1 -9468.412,E2 -9468.412} C_VEL
LIN {X 0,Y 437.206,Z 671.521,A -85,B 0,C 180,E1 -9468.967,E2 -9468.967} C_VEL
LIN {X 0,Y 437.703,Z 656.408,A -85,B 0,C 180,E1 -9469.37,E2 -9469.37} C_VEL
LIN {X 0,Y 439.474,Z 567.091,A -85,B 0,C 180,E1 -9471.112,E2 -9471.112} C_VEL
LIN {X 0,Y 439.852,Z 545.664,A -85,B 0,C 180,E1 -9471.561,E2 -9471.561} C_VEL
LIN {X 0,Y 437.692,Z 531.606,A -85,B 0,C 180,E1 -9472.013,E2 -9472.013} C_VEL
LIN {X 0,Y 436.773,Z 526.756,A -85,B 0,C 180,E1 -9472.203,E2 -9472.203} C_VEL
LIN {X 0,Y 438.794,Z 507.858,A -85,B 0,C 180,E1 -9475.369,E2 -9475.369} C_VEL
LIN {X 0,Y 437.968,Z 502.172,A -85,B 0,C 180,E1 -9476.499,E2 -9476.499} C_VEL
LIN {X 0,Y 435.883,Z 493.534,A -85,B 0,C 180,E1 -9478.402,E2 -9478.402} C_VEL
LIN {X 0,Y 433.125,Z 484.354,A -85,B 0,C 180,E1 -9480.684,E2 -9480.684} C_VEL
LIN {X 0,Y 432.324,Z 481.762,A -85,B 0,C 180,E1 -9481.405,E2 -9481.405} C_VEL
LIN {X 0,Y 432.342,Z 481.758,A -85,B 0,C 180,E1 -9484.677,E2 -9484.677} C_VEL
LIN {X 0,Y 432.341,Z 481.757,A -85,B 0,C 180,E1 -9488.15,E2 -9488.15} C_VEL
LIN {X 0,Y 432.337,Z 481.758,A -85,B 0,C 180,E1 -9491.602,E2 -9491.602} C_VEL
LIN {X 0,Y 432.343,Z 481.755,A -85,B 0,C 180,E1 -9494.346,E2 -9494.346} C_VEL
LIN {X 0,Y 432.323,Z 481.759,A -85,B 0,C 180,E1 -9497.016,E2 -9497.016} C_VEL
LIN {X 0,Y 432.339,Z 481.757,A -85,B 0,C 180,E1 -9499.82,E2 -9499.82} C_VEL
LIN {X 0,Y 432.31,Z 481.762,A -85,B 0,C 180,E1 -9503.022,E2 -9503.022} C_VEL
LIN {X 0,Y 432.362,Z 481.755,A -85,B 0,C 180,E1 -9505.997,E2 -9505.997} C_VEL
LIN {X 0,Y 432.355,Z 481.816,A -85,B 0,C 180,E1 -9509.415,E2 -9509.415} C_VEL
LIN {X 0,Y 435.255,Z 491.607,A -85,B 0,C 180,E1 -9512.079,E2 -9512.079} C_VEL
LIN {X 0,Y 437.397,Z 501.496,A -85,B 0,C 180,E1 -9514.44,E2 -9514.44} C_VEL
LIN {X 0,Y 438.059,Z 505.61,A -85,B 0,C 180,E1 -9515.346,E2 -9515.346} C_VEL
LIN {X 0,Y 436.048,Z 526.098,A -85,B 0,C 180,E1 -9519.232,E2 -9519.232} C_VEL
LIN {X 0,Y 435.052,Z 539.826,A -85,B 0,C 180,E1 -9521.729,E2 -9521.729} C_VEL
LIN {X 0,Y 438.423,Z 557.889,A -85,B 0,C 180,E1 -9522.394,E2 -9522.394} C_VEL
LIN {X 0,Y 439.034,Z 563.528,A -85,B 0,C 180,E1 -9522.572,E2 -9522.572} C_VEL
LIN {X 0,Y 436.835,Z 644.948,A -85,B 0,C 180,E1 -9524.367,E2 -9524.367} C_VEL
LIN {X 0,Y 436.423,Z 659.109,A -85,B 0,C 180,E1 -9524.74,E2 -9524.74} C_VEL
LIN {X 0,Y 435.876,Z 673.57,A -85,B 0,C 180,E1 -9525.338,E2 -9525.338} C_VEL
LIN {X 0,Y 435.4,Z 685.003,A -85,B 0,C 180,E1 -9525.988,E2 -9525.988} C_VEL
LIN {X 0,Y 434.788,Z 696.249,A -85,B 0,C 180,E1 -9526.802,E2 -9526.802} C_VEL
LIN {X 0,Y 433.925,Z 707.834,A -85,B 0,C 180,E1 -9527.845,E2 -9527.845} C_VEL
LIN {X 0,Y 433.361,Z 718.174,A -85,B 0,C 180,E1 -9529.015,E2 -9529.015} C_VEL
LIN {X 0,Y 432.792,Z 728.152,A -85,B 0,C 180,E1 -9530.419,E2 -9530.419} C_VEL
LIN {X 0,Y 432.219,Z 736.208,A -85,B 0,C 180,E1 -9531.82,E2 -9531.82} C_VEL
LIN {X 0,Y 431.947,Z 741.613,A -85,B 0,C 180,E1 -9532.982,E2 -9532.982} C_VEL
LIN {X 0,Y 431.618,Z 746.976,A -85,B 0,C 180,E1 -9534.393,E2 -9534.393} C_VEL
LIN {X 0,Y 431.546,Z 751.089,A -85,B 0,C 180,E1 -9535.797,E2 -9535.797} C_VEL
LIN {X 0,Y 431.373,Z 754.125,A -85,B 0,C 180,E1 -9537.198,E2 -9537.198} C_VEL
LIN {X 0,Y 431.255,Z 755.582,A -85,B 0,C 180,E1 -9538.132,E2 -9538.132} C_VEL
LIN {X 0,Y 431.198,Z 756.601,A -85,B 0,C 180,E1 -9539.066,E2 -9539.066} C_VEL
LIN {X 0,Y 431.168,Z 757.215,A -85,B 0,C 180,E1 -9540,E2 -9540} C_VEL
LIN {X 0,Y 431.172,Z 757.423,A -85,B 0,C 180,E1 -9540.934,E2 -9540.934} C_VEL
LIN {X 0,Y 431.224,Z 757.174,A -85,B 0,C 180,E1 -9541.868,E2 -9541.868} C_VEL
LIN {X 0,Y 431.291,Z 756.509,A -85,B 0,C 180,E1 -9542.802,E2 -9542.802} C_VEL
LIN {X 0,Y 431.247,Z 755.44,A -85,B 0,C 180,E1 -9543.738,E2 -9543.738} C_VEL
LIN {X 0,Y 431.293,Z 753.946,A -85,B 0,C 180,E1 -9544.673,E2 -9544.673} C_VEL
LIN {X 0,Y 431.393,Z 750.76,A -85,B 0,C 180,E1 -9546.107,E2 -9546.107} C_VEL
LIN {X 0,Y 431.536,Z 746.63,A -85,B 0,C 180,E1 -9547.486,E2 -9547.486} C_VEL
LIN {X 0,Y 431.829,Z 740.16,A -85,B 0,C 180,E1 -9549.13,E2 -9549.13} C_VEL
LIN {X 0,Y 432.163,Z 733.116,A -85,B 0,C 180,E1 -9550.542,E2 -9550.542} C_VEL
LIN {X 0,Y 432.742,Z 724.343,A -85,B 0,C 180,E1 -9551.951,E2 -9551.951} C_VEL
LIN {X 0,Y 433.189,Z 714.415,A -85,B 0,C 180,E1 -9553.236,E2 -9553.236} C_VEL
LIN {X 0,Y 433.801,Z 704.247,A -85,B 0,C 180,E1 -9554.304,E2 -9554.304} C_VEL
LIN {X 0,Y 434.476,Z 693.172,A -85,B 0,C 180,E1 -9555.24,E2 -9555.24} C_VEL
LIN {X 0,Y 434.992,Z 680.878,A -85,B 0,C 180,E1 -9556.062,E2 -9556.062} C_VEL
LIN {X 0,Y 435.458,Z 668.198,A -85,B 0,C 180,E1 -9556.707,E2 -9556.707} C_VEL
LIN {X 0,Y 435.945,Z 655,A -85,B 0,C 180,E1 -9557.171,E2 -9557.171} C_VEL
LIN {X 0,Y 436.325,Z 635.953,A -85,B 0,C 180,E1 -9557.578,E2 -9557.578} C_VEL
LIN {X 0,Y 437.562,Z 561.409,A -85,B 0,C 180,E1 -9559.042,E2 -9559.042} C_VEL
LIN {X 0,Y 434.274,Z 540.502,A -85,B 0,C 180,E1 -9559.621,E2 -9559.621} C_VEL
LIN {X 0,Y 435.526,Z 519.115,A -85,B 0,C 180,E1 -9563.356,E2 -9563.356} C_VEL
LIN {X 0,Y 436.66,Z 502.624,A -85,B 0,C 180,E1 -9566.271,E2 -9566.271} C_VEL
LIN {X 0,Y 435.838,Z 497.248,A -85,B 0,C 180,E1 -9567.299,E2 -9567.299} C_VEL
LIN {X 0,Y 432.815,Z 483.944,A -85,B 0,C 180,E1 -9569.955,E2 -9569.955} C_VEL
LIN {X 0,Y 432.34,Z 481.758,A -85,B 0,C 180,E1 -9570.419,E2 -9570.419} C_VEL
LIN {X 0,Y 432.362,Z 481.755,A -85,B 0,C 180,E1 -9574.003,E2 -9574.003} C_VEL
LIN {X 0,Y 432.334,Z 481.755,A -85,B 0,C 180,E1 -9577.198,E2 -9577.198} C_VEL
LIN {X 0,Y 432.343,Z 481.752,A -85,B 0,C 180,E1 -9580.18,E2 -9580.18} C_VEL
LIN {X 0,Y 432.319,Z 481.756,A -85,B 0,C 180,E1 -9583.061,E2 -9583.061} C_VEL
LIN {X 0,Y 432.335,Z 481.759,A -85,B 0,C 180,E1 -9585.665,E2 -9585.665} C_VEL
LIN {X 0,Y 432.334,Z 481.752,A -85,B 0,C 180,E1 -9588.398,E2 -9588.398} C_VEL
LIN {X 0,Y 432.337,Z 481.756,A -85,B 0,C 180,E1 -9591.85,E2 -9591.85} C_VEL
LIN {X 0,Y 432.342,Z 481.756,A -85,B 0,C 180,E1 -9595.323,E2 -9595.323} C_VEL
LIN {X 0,Y 432.323,Z 481.754,A -85,B 0,C 180,E1 -9598.654,E2 -9598.654} C_VEL
LIN {X 0,Y 432.383,Z 481.749,A -85,B 0,C 180,E1 -9601.877,E2 -9601.877} C_VEL
LIN {X 0,Y 432.353,Z 481.752,A -85,B 0,C 180,E1 -9604.999,E2 -9604.999} C_VEL
LIN {X 0,Y 432.359,Z 481.751,A -85,B 0,C 180,E1 -9608.046,E2 -9608.046} C_VEL
LIN {X 0,Y 432.389,Z 481.747,A -85,B 0,C 180,E1 -9611.03,E2 -9611.03} C_VEL
LIN {X 0,Y 432.433,Z 481.742,A -85,B 0,C 180,E1 -9613.961,E2 -9613.961} C_VEL
LIN {X 0,Y 432.374,Z 481.749,A -85,B 0,C 180,E1 -9616.073,E2 -9616.073} C_VEL
LIN {X 0,Y 431.704,Z 481.833,A -85,B 0,C 180,E1 -9616.851,E2 -9616.851} C_VEL
LIN {X 0,Y 428.845,Z 482.188,A -85,B 0,C 180,E1 -9618.115,E2 -9618.115} C_VEL
LIN {X 0,Y 426.448,Z 482.489,A -85,B 0,C 180,E1 -9619.135,E2 -9619.135} C_VEL
LIN {X 0,Y 425.446,Z 482.613,A -85,B 0,C 180,E1 -9619.923,E2 -9619.923} C_VEL
LIN {X 0,Y 425.38,Z 482.619,A -85,B 0,C 180,E1 -9620.19,E2 -9620.19} C_VEL
LIN {X 0,Y 425.539,Z 482.599,A -85,B 0,C 180,E1 -9622.408,E2 -9622.408} C_VEL
LIN {X 0,Y 425.556,Z 482.597,A -85,B 0,C 180,E1 -9624.313,E2 -9624.313} C_VEL
LIN {X 0,Y 425.577,Z 482.595,A -85,B 0,C 180,E1 -9628.107,E2 -9628.107} C_VEL
LIN {X 0,Y 425.705,Z 482.579,A -85,B 0,C 180,E1 -9630,E2 -9630} C_VEL
LIN {X 0,Y 425.559,Z 482.597,A -85,B 0,C 180,E1 -9632.84,E2 -9632.84} C_VEL
LIN {X 0,Y 425.529,Z 482.6,A -85,B 0,C 180,E1 -9636.639,E2 -9636.639} C_VEL
LIN {X 0,Y 425.403,Z 482.622,A -85,B 0,C 180,E1 -9639.509,E2 -9639.509} C_VEL
LIN {X 0,Y 425.395,Z 482.618,A -85,B 0,C 180,E1 -9642.904,E2 -9642.904} C_VEL
LIN {X 0,Y 425.363,Z 482.621,A -85,B 0,C 180,E1 -9646.605,E2 -9646.605} C_VEL
LIN {X 0,Y 425.33,Z 482.629,A -85,B 0,C 180,E1 -9649.636,E2 -9649.636} C_VEL
LIN {X 0,Y 425.309,Z 482.635,A -85,B 0,C 180,E1 -9653.365,E2 -9653.365} C_VEL
LIN {X 0,Y 425.35,Z 482.624,A -85,B 0,C 180,E1 -9656.844,E2 -9656.844} C_VEL
LIN {X 0,Y 425.292,Z 482.633,A -85,B 0,C 180,E1 -9659.72,E2 -9659.72} C_VEL
LIN {X 0,Y 425.283,Z 482.634,A -85,B 0,C 180,E1 -9663.048,E2 -9663.048} C_VEL
LIN {X 0,Y 425.283,Z 482.632,A -85,B 0,C 180,E1 -9665.929,E2 -9665.929} C_VEL
LIN {X 0,Y 425.302,Z 482.632,A -85,B 0,C 180,E1 -9669.044,E2 -9669.044} C_VEL
LIN {X 0,Y 425.28,Z 482.632,A -85,B 0,C 180,E1 -9672.653,E2 -9672.653} C_VEL
LIN {X 0,Y 425.263,Z 482.634,A -85,B 0,C 180,E1 -9676.044,E2 -9676.044} C_VEL
LIN {X 0,Y 425.276,Z 482.632,A -85,B 0,C 180,E1 -9678.622,E2 -9678.622} C_VEL
LIN {X 0,Y 425.308,Z 482.633,A -85,B 0,C 180,E1 -9681.102,E2 -9681.102} C_VEL
LIN {X 0,Y 425.301,Z 482.629,A -85,B 0,C 180,E1 -9684.664,E2 -9684.664} C_VEL
LIN {X 0,Y 425.267,Z 482.634,A -85,B 0,C 180,E1 -9688.073,E2 -9688.073} C_VEL
LIN {X 0,Y 425.343,Z 482.637,A -85,B 0,C 180,E1 -9691.087,E2 -9691.087} C_VEL
LIN {X 0,Y 428.639,Z 497.74,A -85,B 0,C 180,E1 -9693.724,E2 -9693.724} C_VEL
LIN {X 0,Y 429.338,Z 502.985,A -85,B 0,C 180,E1 -9694.605,E2 -9694.605} C_VEL
LIN {X 0,Y 428.507,Z 521.738,A -85,B 0,C 180,E1 -9697.584,E2 -9697.584} C_VEL
LIN {X 0,Y 427.691,Z 540.551,A -85,B 0,C 180,E1 -9700.564,E2 -9700.564} C_VEL
LIN {X 0,Y 427.441,Z 546.764,A -85,B 0,C 180,E1 -9701.545,E2 -9701.545} C_VEL
LIN {X 0,Y 430.21,Z 565.045,A -85,B 0,C 180,E1 -9702.033,E2 -9702.033} C_VEL
LIN {X 0,Y 428.756,Z 656.999,A -85,B 0,C 180,E1 -9703.85,E2 -9703.85} C_VEL
LIN {X 0,Y 428.344,Z 670.356,A -85,B 0,C 180,E1 -9704.293,E2 -9704.293} C_VEL
LIN {X 0,Y 427.81,Z 683.591,A -85,B 0,C 180,E1 -9704.944,E2 -9704.944} C_VEL
LIN {X 0,Y 427.291,Z 695.393,A -85,B 0,C 180,E1 -9705.717,E2 -9705.717} C_VEL
LIN {X 0,Y 426.775,Z 706.701,A -85,B 0,C 180,E1 -9706.671,E2 -9706.671} C_VEL
LIN {X 0,Y 426.126,Z 718.004,A -85,B 0,C 180,E1 -9707.861,E2 -9707.861} C_VEL
LIN {X 0,Y 425.598,Z 727.075,A -85,B 0,C 180,E1 -9709.053,E2 -9709.053} C_VEL
LIN {X 0,Y 425.094,Z 735.933,A -85,B 0,C 180,E1 -9710.484,E2 -9710.484} C_VEL
LIN {X 0,Y 424.706,Z 743.006,A -85,B 0,C 180,E1 -9711.914,E2 -9711.914} C_VEL
LIN {X 0,Y 424.5,Z 748.796,A -85,B 0,C 180,E1 -9713.394,E2 -9713.394} C_VEL
LIN {X 0,Y 424.351,Z 753.015,A -85,B 0,C 180,E1 -9714.774,E2 -9714.774} C_VEL
LIN {X 0,Y 424.19,Z 756.291,A -85,B 0,C 180,E1 -9716.2,E2 -9716.2} C_VEL
LIN {X 0,Y 424.2,Z 757.915,A -85,B 0,C 180,E1 -9717.151,E2 -9717.151} C_VEL
LIN {X 0,Y 424.151,Z 759.088,A -85,B 0,C 180,E1 -9718.101,E2 -9718.101} C_VEL
LIN {X 0,Y 424.091,Z 759.817,A -85,B 0,C 180,E1 -9719.05,E2 -9719.05} C_VEL
LIN {X 0,Y 424.084,Z 760.145,A -85,B 0,C 180,E1 -9720,E2 -9720} C_VEL
LIN {X 0,Y 424.091,Z 760.055,A -85,B 0,C 180,E1 -9720.95,E2 -9720.95} C_VEL
LIN {X 0,Y 424.152,Z 759.502,A -85,B 0,C 180,E1 -9721.899,E2 -9721.899} C_VEL
LIN {X 0,Y 424.253,Z 758.543,A -85,B 0,C 180,E1 -9722.849,E2 -9722.849} C_VEL
LIN {X 0,Y 424.22,Z 757.175,A -85,B 0,C 180,E1 -9723.8,E2 -9723.8} C_VEL
LIN {X 0,Y 424.366,Z 754.243,A -85,B 0,C 180,E1 -9725.226,E2 -9725.226} C_VEL
LIN {X 0,Y 424.583,Z 750.059,A -85,B 0,C 180,E1 -9726.702,E2 -9726.702} C_VEL
LIN {X 0,Y 424.862,Z 743.972,A -85,B 0,C 180,E1 -9728.322,E2 -9728.322} C_VEL
LIN {X 0,Y 425.324,Z 737.16,A -85,B 0,C 180,E1 -9729.751,E2 -9729.751} C_VEL
LIN {X 0,Y 425.843,Z 728.613,A -85,B 0,C 180,E1 -9731.182,E2 -9731.182} C_VEL
LIN {X 0,Y 426.428,Z 719.847,A -85,B 0,C 180,E1 -9732.372,E2 -9732.372} C_VEL
LIN {X 0,Y 427.105,Z 709.458,A -85,B 0,C 180,E1 -9733.519,E2 -9733.519} C_VEL
LIN {X 0,Y 427.721,Z 698.204,A -85,B 0,C 180,E1 -9734.512,E2 -9734.512} C_VEL
LIN {X 0,Y 428.257,Z 686.279,A -85,B 0,C 180,E1 -9735.345,E2 -9735.345} C_VEL
LIN {X 0,Y 428.9,Z 673.798,A -85,B 0,C 180,E1 -9735.991,E2 -9735.991} C_VEL
LIN {X 0,Y 429.36,Z 660.333,A -85,B 0,C 180,E1 -9736.493,E2 -9736.493} C_VEL
LIN {X 0,Y 429.852,Z 633.402,A -85,B 0,C 180,E1 -9737.085,E2 -9737.085} C_VEL
LIN {X 0,Y 431.466,Z 565.553,A -85,B 0,C 180,E1 -9738.541,E2 -9738.541} C_VEL
LIN {X 0,Y 428.853,Z 549.968,A -85,B 0,C 180,E1 -9739.078,E2 -9739.078} C_VEL
LIN {X 0,Y 428.492,Z 548.165,A -85,B 0,C 180,E1 -9739.15,E2 -9739.15} C_VEL
LIN {X 0,Y 429.492,Z 525.965,A -85,B 0,C 180,E1 -9742.615,E2 -9742.615} C_VEL
LIN {X 0,Y 430.523,Z 505.222,A -85,B 0,C 180,E1 -9745.851,E2 -9745.851} C_VEL
LIN {X 0,Y 429.868,Z 500.031,A -85,B 0,C 180,E1 -9746.718,E2 -9746.718} C_VEL
LIN {X 0,Y 427.639,Z 490.384,A -85,B 0,C 180,E1 -9748.464,E2 -9748.464} C_VEL
LIN {X 0,Y 425.313,Z 482.635,A -85,B 0,C 180,E1 -9749.991,E2 -9749.991} C_VEL
LIN {X 0,Y 425.284,Z 482.638,A -85,B 0,C 180,E1 -9753.048,E2 -9753.048} C_VEL
LIN {X 0,Y 425.284,Z 482.635,A -85,B 0,C 180,E1 -9755.929,E2 -9755.929} C_VEL
LIN {X 0,Y 425.3,Z 482.634,A -85,B 0,C 180,E1 -9759.043,E2 -9759.043} C_VEL
LIN {X 0,Y 425.277,Z 482.637,A -85,B 0,C 180,E1 -9762.653,E2 -9762.653} C_VEL
LIN {X 0,Y 425.27,Z 482.635,A -85,B 0,C 180,E1 -9766.045,E2 -9766.045} C_VEL
LIN {X 0,Y 425.3,Z 482.633,A -85,B 0,C 180,E1 -9768.624,E2 -9768.624} C_VEL
LIN {X 0,Y 425.317,Z 482.629,A -85,B 0,C 180,E1 -9771.103,E2 -9771.103} C_VEL
LIN {X 0,Y 425.302,Z 482.632,A -85,B 0,C 180,E1 -9774.664,E2 -9774.664} C_VEL
LIN {X 0,Y 425.276,Z 482.636,A -85,B 0,C 180,E1 -9778.074,E2 -9778.074} C_VEL
LIN {X 0,Y 425.363,Z 482.701,A -85,B 0,C 180,E1 -9780.585,E2 -9780.585} C_VEL
LIN {X 0,Y 429.199,Z 498.595,A -85,B 0,C 180,E1 -9783.499,E2 -9783.499} C_VEL
LIN {X 0,Y 430.632,Z 505.311,A -85,B 0,C 180,E1 -9784.682,E2 -9784.682} C_VEL
LIN {X 0,Y 429.227,Z 524.013,A -85,B 0,C 180,E1 -9787.624,E2 -9787.624} C_VEL
LIN {X 0,Y 429.122,Z 525.598,A -85,B 0,C 180,E1 -9787.871,E2 -9787.871} C_VEL
LIN {X 0,Y 432.449,Z 547.071,A -85,B 0,C 180,E1 -9788.457,E2 -9788.457} C_VEL
LIN {X 0,Y 430.346,Z 662.421,A -85,B 0,C 180,E1 -9790.658,E2 -9790.658} C_VEL
LIN {X 0,Y 429.809,Z 677.067,A -85,B 0,C 180,E1 -9791.128,E2 -9791.128} C_VEL
LIN {X 0,Y 429.275,Z 690.057,A -85,B 0,C 180,E1 -9791.726,E2 -9791.726} C_VEL
LIN {X 0,Y 428.634,Z 702.414,A -85,B 0,C 180,E1 -9792.465,E2 -9792.465} C_VEL
LIN {X 0,Y 427.854,Z 715.038,A -85,B 0,C 180,E1 -9793.417,E2 -9793.417} C_VEL
LIN {X 0,Y 427.065,Z 726.565,A -85,B 0,C 180,E1 -9794.489,E2 -9794.489} C_VEL
LIN {X 0,Y 426.322,Z 737.143,A -85,B 0,C 180,E1 -9795.684,E2 -9795.684} C_VEL
LIN {X 0,Y 425.724,Z 747.231,A -85,B 0,C 180,E1 -9797.061,E2 -9797.061} C_VEL
LIN {X 0,Y 425.215,Z 756.244,A -85,B 0,C 180,E1 -9798.56,E2 -9798.56} C_VEL
LIN {X 0,Y 424.729,Z 764.425,A -85,B 0,C 180,E1 -9800.235,E2 -9800.235} C_VEL
LIN {X 0,Y 424.397,Z 770.972,A -85,B 0,C 180,E1 -9801.908,E2 -9801.908} C_VEL
LIN {X 0,Y 424.232,Z 776.451,A -85,B 0,C 180,E1 -9803.713,E2 -9803.713} C_VEL
LIN {X 0,Y 424.174,Z 779.93,A -85,B 0,C 180,E1 -9805.248,E2 -9805.248} C_VEL
LIN {X 0,Y 424.13,Z 782.87,A -85,B 0,C 180,E1 -9807.151,E2 -9807.151} C_VEL
LIN {X 0,Y 424.141,Z 783.792,A -85,B 0,C 180,E1 -9808.101,E2 -9808.101} C_VEL
LIN {X 0,Y 424.083,Z 784.559,A -85,B 0,C 180,E1 -9810,E2 -9810} C_VEL
LIN {X 0,Y 424.141,Z 783.893,A -85,B 0,C 180,E1 -9811.899,E2 -9811.899} C_VEL
LIN {X 0,Y 424.09,Z 781.762,A -85,B 0,C 180,E1 -9813.801,E2 -9813.801} C_VEL
LIN {X 0,Y 424.181,Z 779.205,A -85,B 0,C 180,E1 -9815.228,E2 -9815.228} C_VEL
LIN {X 0,Y 424.316,Z 774.428,A -85,B 0,C 180,E1 -9817.136,E2 -9817.136} C_VEL
LIN {X 0,Y 424.475,Z 769.706,A -85,B 0,C 180,E1 -9818.57,E2 -9818.57} C_VEL
LIN {X 0,Y 424.799,Z 762.875,A -85,B 0,C 180,E1 -9820.245,E2 -9820.245} C_VEL
LIN {X 0,Y 425.385,Z 754.318,A -85,B 0,C 180,E1 -9821.919,E2 -9821.919} C_VEL
LIN {X 0,Y 425.961,Z 745.357,A -85,B 0,C 180,E1 -9823.355,E2 -9823.355} C_VEL
LIN {X 0,Y 426.652,Z 734.479,A -85,B 0,C 180,E1 -9824.793,E2 -9824.793} C_VEL
LIN {X 0,Y 427.458,Z 723.462,A -85,B 0,C 180,E1 -9825.986,E2 -9825.986} C_VEL
LIN {X 0,Y 428.305,Z 711.434,A -85,B 0,C 180,E1 -9827.056,E2 -9827.056} C_VEL
LIN {X 0,Y 429.199,Z 698.094,A -85,B 0,C 180,E1 -9828.004,E2 -9828.004} C_VEL
LIN {X 0,Y 429.927,Z 684.463,A -85,B 0,C 180,E1 -9828.75,E2 -9828.75} C_VEL
LIN {X 0,Y 430.563,Z 670.842,A -85,B 0,C 180,E1 -9829.302,E2 -9829.302} C_VEL
LIN {X 0,Y 431.033,Z 656.962,A -85,B 0,C 180,E1 -9829.682,E2 -9829.682} C_VEL
LIN {X 0,Y 432.991,Z 568.636,A -85,B 0,C 180,E1 -9831.46,E2 -9831.46} C_VEL
LIN {X 0,Y 433.462,Z 546.96,A -85,B 0,C 180,E1 -9831.927,E2 -9831.927} C_VEL
LIN {X 0,Y 431.405,Z 533.226,A -85,B 0,C 180,E1 -9832.384,E2 -9832.384} C_VEL
LIN {X 0,Y 430.182,Z 526.991,A -85,B 0,C 180,E1 -9832.638,E2 -9832.638} C_VEL
LIN {X 0,Y 432.134,Z 510.118,A -85,B 0,C 180,E1 -9835.53,E2 -9835.53} C_VEL
LIN {X 0,Y 431.41,Z 504.604,A -85,B 0,C 180,E1 -9836.658,E2 -9836.658} C_VEL
LIN {X 0,Y 429.355,Z 496.101,A -85,B 0,C 180,E1 -9838.593,E2 -9838.593} C_VEL
LIN {X 0,Y 426.948,Z 487.955,A -85,B 0,C 180,E1 -9840.684,E2 -9840.684} C_VEL
LIN {X 0,Y 425.285,Z 482.637,A -85,B 0,C 180,E1 -9842.256,E2 -9842.256} C_VEL
LIN {X 0,Y 425.301,Z 482.636,A -85,B 0,C 180,E1 -9845.336,E2 -9845.336} C_VEL
LIN {X 0,Y 425.3,Z 482.635,A -85,B 0,C 180,E1 -9849.044,E2 -9849.044} C_VEL
LIN {X 0,Y 425.281,Z 482.636,A -85,B 0,C 180,E1 -9852.653,E2 -9852.653} C_VEL
LIN {X 0,Y 425.264,Z 482.637,A -85,B 0,C 180,E1 -9856.044,E2 -9856.044} C_VEL
LIN {X 0,Y 425.277,Z 482.638,A -85,B 0,C 180,E1 -9858.622,E2 -9858.622} C_VEL
LIN {X 0,Y 425.313,Z 482.633,A -85,B 0,C 180,E1 -9861.103,E2 -9861.103} C_VEL
LIN {X 0,Y 425.302,Z 482.635,A -85,B 0,C 180,E1 -9864.664,E2 -9864.664} C_VEL
LIN {X 0,Y 425.268,Z 482.639,A -85,B 0,C 180,E1 -9868.073,E2 -9868.073} C_VEL
LIN {X 0,Y 425.314,Z 482.764,A -85,B 0,C 180,E1 -9868.634,E2 -9868.634} C_VEL
LIN {X 0,Y 427.702,Z 490.638,A -85,B 0,C 180,E1 -9870.952,E2 -9870.952} C_VEL
LIN {X 0,Y 429.736,Z 498.51,A -85,B 0,C 180,E1 -9873.01,E2 -9873.01} C_VEL
LIN {X 0,Y 431.274,Z 506.639,A -85,B 0,C 180,E1 -9874.932,E2 -9874.932} C_VEL
LIN {X 0,Y 431.088,Z 510.351,A -85,B 0,C 180,E1 -9875.691,E2 -9875.691} C_VEL
LIN {X 0,Y 429.261,Z 528.247,A -85,B 0,C 180,E1 -9879.144,E2 -9879.144} C_VEL
LIN {X 0,Y 428.383,Z 539.828,A -85,B 0,C 180,E1 -9881.275,E2 -9881.275} C_VEL
LIN {X 0,Y 431.842,Z 557.989,A -85,B 0,C 180,E1 -9881.988,E2 -9881.988} C_VEL
LIN {X 0,Y 432.565,Z 564.153,A -85,B 0,C 180,E1 -9882.197,E2 -9882.197} C_VEL
LIN {X 0,Y 429.911,Z 654.992,A -85,B 0,C 180,E1 -9884.291,E2 -9884.291} C_VEL
LIN {X 0,Y 429.351,Z 669.104,A -85,B 0,C 180,E1 -9884.817,E2 -9884.817} C_VEL
LIN {X 0,Y 428.766,Z 682.17,A -85,B 0,C 180,E1 -9885.519,E2 -9885.519} C_VEL
LIN {X 0,Y 428.097,Z 694.188,A -85,B 0,C 180,E1 -9886.35,E2 -9886.35} C_VEL
LIN {X 0,Y 427.368,Z 705.042,A -85,B 0,C 180,E1 -9887.294,E2 -9887.294} C_VEL
LIN {X 0,Y 426.67,Z 714.959,A -85,B 0,C 180,E1 -9888.359,E2 -9888.359} C_VEL
LIN {X 0,Y 426.138,Z 724.022,A -85,B 0,C 180,E1 -9889.548,E2 -9889.548} C_VEL
LIN {X 0,Y 425.455,Z 732.923,A -85,B 0,C 180,E1 -9890.971,E2 -9890.971} C_VEL
LIN {X 0,Y 425.008,Z 740.024,A -85,B 0,C 180,E1 -9892.398,E2 -9892.398} C_VEL
LIN {X 0,Y 424.77,Z 745.713,A -85,B 0,C 180,E1 -9893.826,E2 -9893.826} C_VEL
LIN {X 0,Y 424.402,Z 750.193,A -85,B 0,C 180,E1 -9895.251,E2 -9895.251} C_VEL
LIN {X 0,Y 424.454,Z 752.546,A -85,B 0,C 180,E1 -9896.202,E2 -9896.202} C_VEL
LIN {X 0,Y 424.31,Z 754.461,A -85,B 0,C 180,E1 -9897.152,E2 -9897.152} C_VEL
LIN {X 0,Y 424.181,Z 755.887,A -85,B 0,C 180,E1 -9898.101,E2 -9898.101} C_VEL
LIN {X 0,Y 424.116,Z 756.888,A -85,B 0,C 180,E1 -9899.05,E2 -9899.05} C_VEL
LIN {X 0,Y 424.085,Z 757.482,A -85,B 0,C 180,E1 -9900,E2 -9900} C_VEL
LIN {X 0,Y 424.091,Z 757.657,A -85,B 0,C 180,E1 -9900.95,E2 -9900.95} C_VEL
LIN {X 0,Y 424.15,Z 757.373,A -85,B 0,C 180,E1 -9901.899,E2 -9901.899} C_VEL
LIN {X 0,Y 424.204,Z 756.682,A -85,B 0,C 180,E1 -9902.849,E2 -9902.849} C_VEL
LIN {X 0,Y 424.154,Z 755.586,A -85,B 0,C 180,E1 -9903.8,E2 -9903.8} C_VEL
LIN {X 0,Y 424.257,Z 753.095,A -85,B 0,C 180,E1 -9905.227,E2 -9905.227} C_VEL
LIN {X 0,Y 424.371,Z 748.997,A -85,B 0,C 180,E1 -9906.848,E2 -9906.848} C_VEL
LIN {X 0,Y 424.543,Z 744.913,A -85,B 0,C 180,E1 -9908.089,E2 -9908.089} C_VEL
LIN {X 0,Y 424.838,Z 738.995,A -85,B 0,C 180,E1 -9909.522,E2 -9909.522} C_VEL
LIN {X 0,Y 425.208,Z 731.563,A -85,B 0,C 180,E1 -9910.957,E2 -9910.957} C_VEL
LIN {X 0,Y 425.83,Z 722.334,A -85,B 0,C 180,E1 -9912.389,E2 -9912.389} C_VEL
LIN {X 0,Y 426.312,Z 712.853,A -85,B 0,C 180,E1 -9913.587,E2 -9913.587} C_VEL
LIN {X 0,Y 426.923,Z 702.333,A -85,B 0,C 180,E1 -9914.661,E2 -9914.661} C_VEL
LIN {X 0,Y 427.596,Z 690.755,A -85,B 0,C 180,E1 -9915.613,E2 -9915.613} C_VEL
LIN {X 0,Y 428.198,Z 678.836,A -85,B 0,C 180,E1 -9916.385,E2 -9916.385} C_VEL
LIN {X 0,Y 428.585,Z 665.914,A -85,B 0,C 180,E1 -9917.014,E2 -9917.014} C_VEL
LIN {X 0,Y 429.078,Z 652.809,A -85,B 0,C 180,E1 -9917.454,E2 -9917.454} C_VEL
LIN {X 0,Y 430.71,Z 561.854,A -85,B 0,C 180,E1 -9919.309,E2 -9919.309} C_VEL
LIN {X 0,Y 427.397,Z 540.391,A -85,B 0,C 180,E1 -9919.919,E2 -9919.919} C_VEL
LIN {X 0,Y 428.655,Z 519.151,A -85,B 0,C 180,E1 -9923.683,E2 -9923.683} C_VEL
LIN {X 0,Y 429.77,Z 503.669,A -85,B 0,C 180,E1 -9926.463,E2 -9926.463} C_VEL
LIN {X 0,Y 427.823,Z 493.601,A -85,B 0,C 180,E1 -9928.45,E2 -9928.45} C_VEL
LIN {X 0,Y 425.314,Z 482.633,A -85,B 0,C 180,E1 -9930.708,E2 -9930.708} C_VEL
LIN {X 0,Y 425.314,Z 482.631,A -85,B 0,C 180,E1 -9934.288,E2 -9934.288} C_VEL
LIN {X 0,Y 425.288,Z 482.636,A -85,B 0,C 180,E1 -9937.693,E2 -9937.693} C_VEL
LIN {X 0,Y 425.286,Z 482.63,A -85,B 0,C 180,E1 -9940.521,E2 -9940.521} C_VEL
LIN {X 0,Y 425.26,Z 482.638,A -85,B 0,C 180,E1 -9943.351,E2 -9943.351} C_VEL
LIN {X 0,Y 425.259,Z 482.633,A -85,B 0,C 180,E1 -9946.649,E2 -9946.649} C_VEL
LIN {X 0,Y 425.287,Z 482.634,A -85,B 0,C 180,E1 -9949.872,E2 -9949.872} C_VEL
LIN {X 0,Y 425.279,Z 482.631,A -85,B 0,C 180,E1 -9952.488,E2 -9952.488} C_VEL
LIN {X 0,Y 425.309,Z 482.632,A -85,B 0,C 180,E1 -9955.817,E2 -9955.817} C_VEL
LIN {X 0,Y 425.292,Z 482.633,A -85,B 0,C 180,E1 -9959.239,E2 -9959.239} C_VEL
LIN {X 0,Y 425.35,Z 482.622,A -85,B 0,C 180,E1 -9962.442,E2 -9962.442} C_VEL
LIN {X 0,Y 425.353,Z 482.629,A -85,B 0,C 180,E1 -9965.602,E2 -9965.602} C_VEL
LIN {X 0,Y 425.295,Z 482.629,A -85,B 0,C 180,E1 -9968.681,E2 -9968.681} C_VEL
LIN {X 0,Y 425.335,Z 482.629,A -85,B 0,C 180,E1 -9971.703,E2 -9971.703} C_VEL
LIN {X 0,Y 425.351,Z 482.622,A -85,B 0,C 180,E1 -9974.671,E2 -9974.671} C_VEL
LIN {X 0,Y 425.414,Z 482.62,A -85,B 0,C 180,E1 -9977.598,E2 -9977.598} C_VEL
LIN {X 0,Y 425.38,Z 482.619,A -85,B 0,C 180,E1 -9980.19,E2 -9980.19} C_VEL
LIN {X 0,Y 424.791,Z 482.695,A -85,B 0,C 180,E1 -9980.98,E2 -9980.98} C_VEL
LIN {X 0,Y 422.087,Z 483.029,A -85,B 0,C 180,E1 -9982.268,E2 -9982.268} C_VEL
LIN {X 0,Y 419.713,Z 483.33,A -85,B 0,C 180,E1 -9983.306,E2 -9983.306} C_VEL
LIN {X 0,Y 418.611,Z 483.463,A -85,B 0,C 180,E1 -9984.107,E2 -9984.107} C_VEL
LIN {X 0,Y 418.478,Z 483.478,A -85,B 0,C 180,E1 -9984.379,E2 -9984.379} C_VEL
LIN {X 0,Y 418.546,Z 483.471,A -85,B 0,C 180,E1 -9988.075,E2 -9988.075} C_VEL
LIN {X 0,Y 418.675,Z 483.455,A -85,B 0,C 180,E1 -9990,E2 -9990} C_VEL
LIN {X 0,Y 418.513,Z 483.475,A -85,B 0,C 180,E1 -9992.888,E2 -9992.888} C_VEL
LIN {X 0,Y 418.493,Z 483.477,A -85,B 0,C 180,E1 -9996.751,E2 -9996.751} C_VEL
LIN {X 0,Y 418.402,Z 483.488,A -85,B 0,C 180,E1 -9998.695,E2 -9998.695} C_VEL
LIN {X 0,Y 418.318,Z 483.503,A -85,B 0,C 180,E1 -10001.631,E2 -10001.631} C_VEL
LIN {X 0,Y 418.306,Z 483.5,A -85,B 0,C 180,E1 -10004.597,E2 -10004.597} C_VEL
LIN {X 0,Y 418.29,Z 483.507,A -85,B 0,C 180,E1 -10007.604,E2 -10007.604} C_VEL
LIN {X 0,Y 418.252,Z 483.507,A -85,B 0,C 180,E1 -10010.663,E2 -10010.663} C_VEL
LIN {X 0,Y 418.29,Z 483.504,A -85,B 0,C 180,E1 -10013.781,E2 -10013.781} C_VEL
LIN {X 0,Y 418.311,Z 483.503,A -85,B 0,C 180,E1 -10017.071,E2 -10017.071} C_VEL
LIN {X 0,Y 418.246,Z 483.507,A -85,B 0,C 180,E1 -10020.272,E2 -10020.272} C_VEL
LIN {X 0,Y 418.25,Z 483.51,A -85,B 0,C 180,E1 -10023.677,E2 -10023.677} C_VEL
LIN {X 0,Y 418.242,Z 483.514,A -85,B 0,C 180,E1 -10027.224,E2 -10027.224} C_VEL
LIN {X 0,Y 418.256,Z 483.509,A -85,B 0,C 180,E1 -10029.682,E2 -10029.682} C_VEL
LIN {X 0,Y 418.234,Z 483.509,A -85,B 0,C 180,E1 -10032.322,E2 -10032.322} C_VEL
LIN {X 0,Y 418.24,Z 483.513,A -85,B 0,C 180,E1 -10035.109,E2 -10035.109} C_VEL
LIN {X 0,Y 418.241,Z 483.51,A -85,B 0,C 180,E1 -10037.767,E2 -10037.767} C_VEL
LIN {X 0,Y 418.254,Z 483.507,A -85,B 0,C 180,E1 -10040.619,E2 -10040.619} C_VEL
LIN {X 0,Y 418.245,Z 483.508,A -85,B 0,C 180,E1 -10043.976,E2 -10043.976} C_VEL
LIN {X 0,Y 418.26,Z 483.512,A -85,B 0,C 180,E1 -10047.156,E2 -10047.156} C_VEL
LIN {X 0,Y 418.264,Z 483.562,A -85,B 0,C 180,E1 -10050.838,E2 -10050.838} C_VEL
LIN {X 0,Y 421.582,Z 498.473,A -85,B 0,C 180,E1 -10053.472,E2 -10053.472} C_VEL
LIN {X 0,Y 422.446,Z 503.718,A -85,B 0,C 180,E1 -10054.371,E2 -10054.371} C_VEL
LIN {X 0,Y 421.648,Z 521.349,A -85,B 0,C 180,E1 -10057.199,E2 -10057.199} C_VEL
LIN {X 0,Y 420.814,Z 540.339,A -85,B 0,C 180,E1 -10060.233,E2 -10060.233} C_VEL
LIN {X 0,Y 420.543,Z 547.109,A -85,B 0,C 180,E1 -10061.297,E2 -10061.297} C_VEL
LIN {X 0,Y 423.389,Z 566.375,A -85,B 0,C 180,E1 -10061.815,E2 -10061.815} C_VEL
LIN {X 0,Y 421.82,Z 657.905,A -85,B 0,C 180,E1 -10063.671,E2 -10063.671} C_VEL
LIN {X 0,Y 421.403,Z 670.236,A -85,B 0,C 180,E1 -10064.089,E2 -10064.089} C_VEL
LIN {X 0,Y 420.858,Z 683.533,A -85,B 0,C 180,E1 -10064.751,E2 -10064.751} C_VEL
LIN {X 0,Y 420.298,Z 695.92,A -85,B 0,C 180,E1 -10065.577,E2 -10065.577} C_VEL
LIN {X 0,Y 419.751,Z 707.368,A -85,B 0,C 180,E1 -10066.567,E2 -10066.567} C_VEL
LIN {X 0,Y 419.163,Z 717.566,A -85,B 0,C 180,E1 -10067.656,E2 -10067.656} C_VEL
LIN {X 0,Y 418.592,Z 726.776,A -85,B 0,C 180,E1 -10068.867,E2 -10068.867} C_VEL
LIN {X 0,Y 418.066,Z 735.729,A -85,B 0,C 180,E1 -10070.322,E2 -10070.322} C_VEL
LIN {X 0,Y 417.645,Z 742.911,A -85,B 0,C 180,E1 -10071.776,E2 -10071.776} C_VEL
LIN {X 0,Y 417.401,Z 749.245,A -85,B 0,C 180,E1 -10073.422,E2 -10073.422} C_VEL
LIN {X 0,Y 417.205,Z 754.302,A -85,B 0,C 180,E1 -10075.168,E2 -10075.168} C_VEL
LIN {X 0,Y 417.099,Z 756.376,A -85,B 0,C 180,E1 -10076.135,E2 -10076.135} C_VEL
LIN {X 0,Y 417.101,Z 758.028,A -85,B 0,C 180,E1 -10077.103,E2 -10077.103} C_VEL
LIN {X 0,Y 417.079,Z 759.24,A -85,B 0,C 180,E1 -10078.069,E2 -10078.069} C_VEL
LIN {X 0,Y 417.014,Z 759.99,A -85,B 0,C 180,E1 -10079.034,E2 -10079.034} C_VEL
LIN {X 0,Y 417.004,Z 760.337,A -85,B 0,C 180,E1 -10080,E2 -10080} C_VEL
LIN {X 0,Y 417.014,Z 760.271,A -85,B 0,C 180,E1 -10080.966,E2 -10080.966} C_VEL
LIN {X 0,Y 417.081,Z 759.737,A -85,B 0,C 180,E1 -10081.931,E2 -10081.931} C_VEL
LIN {X 0,Y 417.168,Z 758.79,A -85,B 0,C 180,E1 -10082.897,E2 -10082.897} C_VEL
LIN {X 0,Y 417.13,Z 757.436,A -85,B 0,C 180,E1 -10083.864,E2 -10083.864} C_VEL
LIN {X 0,Y 417.317,Z 754.531,A -85,B 0,C 180,E1 -10085.315,E2 -10085.315} C_VEL
LIN {X 0,Y 417.521,Z 750.549,A -85,B 0,C 180,E1 -10086.767,E2 -10086.767} C_VEL
LIN {X 0,Y 417.852,Z 744.351,A -85,B 0,C 180,E1 -10088.463,E2 -10088.463} C_VEL
LIN {X 0,Y 418.332,Z 737.56,A -85,B 0,C 180,E1 -10089.916,E2 -10089.916} C_VEL
LIN {X 0,Y 418.793,Z 730.619,A -85,B 0,C 180,E1 -10091.127,E2 -10091.127} C_VEL
LIN {X 0,Y 419.398,Z 722.211,A -85,B 0,C 180,E1 -10092.337,E2 -10092.337} C_VEL
LIN {X 0,Y 420.09,Z 711.865,A -85,B 0,C 180,E1 -10093.545,E2 -10093.545} C_VEL
LIN {X 0,Y 420.723,Z 701.749,A -85,B 0,C 180,E1 -10094.511,E2 -10094.511} C_VEL
LIN {X 0,Y 421.271,Z 690.763,A -85,B 0,C 180,E1 -10095.358,E2 -10095.358} C_VEL
LIN {X 0,Y 422.011,Z 677.459,A -85,B 0,C 180,E1 -10096.135,E2 -10096.135} C_VEL
LIN {X 0,Y 422.521,Z 664.685,A -85,B 0,C 180,E1 -10096.674,E2 -10096.674} C_VEL
LIN {X 0,Y 422.896,Z 650.314,A -85,B 0,C 180,E1 -10097.063,E2 -10097.063} C_VEL
LIN {X 0,Y 424.731,Z 575.357,A -85,B 0,C 180,E1 -10098.705,E2 -10098.705} C_VEL
LIN {X 0,Y 424.819,Z 565.315,A -85,B 0,C 180,E1 -10098.946,E2 -10098.946} C_VEL
LIN {X 0,Y 422.126,Z 549.893,A -85,B 0,C 180,E1 -10099.511,E2 -10099.511} C_VEL
LIN {X 0,Y 421.834,Z 548.279,A -85,B 0,C 180,E1 -10099.59,E2 -10099.59} C_VEL
LIN {X 0,Y 422.875,Z 526.81,A -85,B 0,C 180,E1 -10102.989,E2 -10102.989} C_VEL
LIN {X 0,Y 423.893,Z 508.309,A -85,B 0,C 180,E1 -10105.91,E2 -10105.91} C_VEL
LIN {X 0,Y 423.681,Z 504.137,A -85,B 0,C 180,E1 -10106.607,E2 -10106.607} C_VEL
LIN {X 0,Y 421.571,Z 494.49,A -85,B 0,C 180,E1 -10108.367,E2 -10108.367} C_VEL
LIN {X 0,Y 418.277,Z 483.512,A -85,B 0,C 180,E1 -10110.574,E2 -10110.574} C_VEL
LIN {X 0,Y 418.251,Z 483.514,A -85,B 0,C 180,E1 -10113.677,E2 -10113.677} C_VEL
LIN {X 0,Y 418.242,Z 483.512,A -85,B 0,C 180,E1 -10117.224,E2 -10117.224} C_VEL
LIN {X 0,Y 418.253,Z 483.511,A -85,B 0,C 180,E1 -10119.682,E2 -10119.682} C_VEL
LIN {X 0,Y 418.231,Z 483.512,A -85,B 0,C 180,E1 -10122.321,E2 -10122.321} C_VEL
LIN {X 0,Y 418.241,Z 483.51,A -85,B 0,C 180,E1 -10125.109,E2 -10125.109} C_VEL
LIN {X 0,Y 418.259,Z 483.508,A -85,B 0,C 180,E1 -10127.769,E2 -10127.769} C_VEL
LIN {X 0,Y 418.262,Z 483.509,A -85,B 0,C 180,E1 -10130.618,E2 -10130.618} C_VEL
LIN {X 0,Y 418.248,Z 483.512,A -85,B 0,C 180,E1 -10133.976,E2 -10133.976} C_VEL
LIN {X 0,Y 418.262,Z 483.509,A -85,B 0,C 180,E1 -10137.155,E2 -10137.155} C_VEL
LIN {X 0,Y 418.319,Z 483.528,A -85,B 0,C 180,E1 -10140.255,E2 -10140.255} C_VEL
LIN {X 0,Y 422.263,Z 499.851,A -85,B 0,C 180,E1 -10143.296,E2 -10143.296} C_VEL
LIN {X 0,Y 423.653,Z 506.26,A -85,B 0,C 180,E1 -10144.449,E2 -10144.449} C_VEL
LIN {X 0,Y 423.324,Z 512.583,A -85,B 0,C 180,E1 -10145.478,E2 -10145.478} C_VEL
LIN {X 0,Y 422.274,Z 525.721,A -85,B 0,C 180,E1 -10147.567,E2 -10147.567} C_VEL
LIN {X 0,Y 425.668,Z 548.248,A -85,B 0,C 180,E1 -10148.191,E2 -10148.191} C_VEL
LIN {X 0,Y 423.486,Z 662.589,A -85,B 0,C 180,E1 -10150.426,E2 -10150.426} C_VEL
LIN {X 0,Y 422.917,Z 677.028,A -85,B 0,C 180,E1 -10150.9,E2 -10150.9} C_VEL
LIN {X 0,Y 422.304,Z 691.104,A -85,B 0,C 180,E1 -10151.567,E2 -10151.567} C_VEL
LIN {X 0,Y 421.614,Z 704.701,A -85,B 0,C 180,E1 -10152.422,E2 -10152.422} C_VEL
LIN {X 0,Y 420.752,Z 716.756,A -85,B 0,C 180,E1 -10153.379,E2 -10153.379} C_VEL
LIN {X 0,Y 419.909,Z 729.034,A -85,B 0,C 180,E1 -10154.591,E2 -10154.591} C_VEL
LIN {X 0,Y 419.087,Z 740.07,A -85,B 0,C 180,E1 -10155.927,E2 -10155.927} C_VEL
LIN {X 0,Y 418.568,Z 750.003,A -85,B 0,C 180,E1 -10157.392,E2 -10157.392} C_VEL
LIN {X 0,Y 417.991,Z 758.183,A -85,B 0,C 180,E1 -10158.851,E2 -10158.851} C_VEL
LIN {X 0,Y 417.553,Z 765.992,A -85,B 0,C 180,E1 -10160.555,E2 -10160.555} C_VEL
LIN {X 0,Y 417.259,Z 772.191,A -85,B 0,C 180,E1 -10162.256,E2 -10162.256} C_VEL
LIN {X 0,Y 417.131,Z 776.456,A -85,B 0,C 180,E1 -10163.751,E2 -10163.751} C_VEL
LIN {X 0,Y 417.082,Z 779.602,A -85,B 0,C 180,E1 -10165.167,E2 -10165.167} C_VEL
LIN {X 0,Y 417.028,Z 782.582,A -85,B 0,C 180,E1 -10167.102,E2 -10167.102} C_VEL
LIN {X 0,Y 417.067,Z 783.523,A -85,B 0,C 180,E1 -10168.069,E2 -10168.069} C_VEL
LIN {X 0,Y 417.002,Z 784.319,A -85,B 0,C 180,E1 -10170,E2 -10170} C_VEL
LIN {X 0,Y 417.067,Z 783.681,A -85,B 0,C 180,E1 -10171.931,E2 -10171.931} C_VEL
LIN {X 0,Y 417.005,Z 781.572,A -85,B 0,C 180,E1 -10173.866,E2 -10173.866} C_VEL
LIN {X 0,Y 417.084,Z 779.962,A -85,B 0,C 180,E1 -10174.833,E2 -10174.833} C_VEL
LIN {X 0,Y 417.226,Z 775.582,A -85,B 0,C 180,E1 -10176.772,E2 -10176.772} C_VEL
LIN {X 0,Y 417.418,Z 769.539,A -85,B 0,C 180,E1 -10178.716,E2 -10178.716} C_VEL
LIN {X 0,Y 417.769,Z 762.723,A -85,B 0,C 180,E1 -10180.419,E2 -10180.419} C_VEL
LIN {X 0,Y 418.384,Z 754.191,A -85,B 0,C 180,E1 -10182.121,E2 -10182.121} C_VEL
LIN {X 0,Y 418.999,Z 745.241,A -85,B 0,C 180,E1 -10183.582,E2 -10183.582} C_VEL
LIN {X 0,Y 419.755,Z 734.395,A -85,B 0,C 180,E1 -10185.042,E2 -10185.042} C_VEL
LIN {X 0,Y 420.618,Z 723.417,A -85,B 0,C 180,E1 -10186.253,E2 -10186.253} C_VEL
LIN {X 0,Y 421.506,Z 711.429,A -85,B 0,C 180,E1 -10187.34,E2 -10187.34} C_VEL
LIN {X 0,Y 422.464,Z 698.193,A -85,B 0,C 180,E1 -10188.301,E2 -10188.301} C_VEL
LIN {X 0,Y 423.249,Z 684.214,A -85,B 0,C 180,E1 -10189.081,E2 -10189.081} C_VEL
LIN {X 0,Y 423.95,Z 670.438,A -85,B 0,C 180,E1 -10189.646,E2 -10189.646} C_VEL
LIN {X 0,Y 424.457,Z 655.259,A -85,B 0,C 180,E1 -10190.063,E2 -10190.063} C_VEL
LIN {X 0,Y 426.435,Z 573.036,A -85,B 0,C 180,E1 -10191.767,E2 -10191.767} C_VEL
LIN {X 0,Y 427.061,Z 547.776,A -85,B 0,C 180,E1 -10192.328,E2 -10192.328} C_VEL
LIN {X 0,Y 425.027,Z 534.226,A -85,B 0,C 180,E1 -10192.802,E2 -10192.802} C_VEL
LIN {X 0,Y 423.635,Z 527.206,A -85,B 0,C 180,E1 -10193.107,E2 -10193.107} C_VEL
LIN {X 0,Y 425.51,Z 512.485,A -85,B 0,C 180,E1 -10195.694,E2 -10195.694} C_VEL
LIN {X 0,Y 425.353,Z 509.801,A -85,B 0,C 180,E1 -10196.231,E2 -10196.231} C_VEL
LIN {X 0,Y 423.349,Z 500.359,A -85,B 0,C 180,E1 -10198.376,E2 -10198.376} C_VEL
LIN {X 0,Y 420.837,Z 491.79,A -85,B 0,C 180,E1 -10200.621,E2 -10200.621} C_VEL
LIN {X 0,Y 418.246,Z 483.514,A -85,B 0,C 180,E1 -10203.127,E2 -10203.127} C_VEL
LIN {X 0,Y 418.247,Z 483.514,A -85,B 0,C 180,E1 -10206.238,E2 -10206.238} C_VEL
LIN {X 0,Y 418.254,Z 483.512,A -85,B 0,C 180,E1 -10209.682,E2 -10209.682} C_VEL
LIN {X 0,Y 418.235,Z 483.512,A -85,B 0,C 180,E1 -10212.322,E2 -10212.322} C_VEL
LIN {X 0,Y 418.241,Z 483.514,A -85,B 0,C 180,E1 -10215.109,E2 -10215.109} C_VEL
LIN {X 0,Y 418.242,Z 483.512,A -85,B 0,C 180,E1 -10217.767,E2 -10217.767} C_VEL
LIN {X 0,Y 418.258,Z 483.512,A -85,B 0,C 180,E1 -10220.619,E2 -10220.619} C_VEL
LIN {X 0,Y 418.246,Z 483.514,A -85,B 0,C 180,E1 -10223.976,E2 -10223.976} C_VEL
LIN {X 0,Y 418.261,Z 483.512,A -85,B 0,C 180,E1 -10227.156,E2 -10227.156} C_VEL
LIN {X 0,Y 418.271,Z 483.732,A -85,B 0,C 180,E1 -10227.759,E2 -10227.759} C_VEL
LIN {X 0,Y 420.744,Z 491.732,A -85,B 0,C 180,E1 -10230.296,E2 -10230.296} C_VEL
LIN {X 0,Y 422.924,Z 499.818,A -85,B 0,C 180,E1 -10232.539,E2 -10232.539} C_VEL
LIN {X 0,Y 424.678,Z 508.952,A -85,B 0,C 180,E1 -10234.777,E2 -10234.777} C_VEL
LIN {X 0,Y 424.22,Z 514.198,A -85,B 0,C 180,E1 -10235.862,E2 -10235.862} C_VEL
LIN {X 0,Y 422.148,Z 534.252,A -85,B 0,C 180,E1 -10239.791,E2 -10239.791} C_VEL
LIN {X 0,Y 421.723,Z 539.678,A -85,B 0,C 180,E1 -10240.781,E2 -10240.781} C_VEL
LIN {X 0,Y 425.336,Z 558.208,A -85,B 0,C 180,E1 -10241.557,E2 -10241.557} C_VEL
LIN {X 0,Y 426.14,Z 565.193,A -85,B 0,C 180,E1 -10241.801,E2 -10241.801} C_VEL
LIN {X 0,Y 423.616,Z 644.499,A -85,B 0,C 180,E1 -10243.68,E2 -10243.68} C_VEL
LIN {X 0,Y 423.088,Z 659.427,A -85,B 0,C 180,E1 -10244.092,E2 -10244.092} C_VEL
LIN {X 0,Y 422.461,Z 673.972,A -85,B 0,C 180,E1 -10244.723,E2 -10244.723} C_VEL
LIN {X 0,Y 421.766,Z 687.227,A -85,B 0,C 180,E1 -10245.525,E2 -10245.525} C_VEL
LIN {X 0,Y 420.955,Z 699.484,A -85,B 0,C 180,E1 -10246.483,E2 -10246.483} C_VEL
LIN {X 0,Y 420.093,Z 710.445,A -85,B 0,C 180,E1 -10247.561,E2 -10247.561} C_VEL
LIN {X 0,Y 419.361,Z 721.265,A -85,B 0,C 180,E1 -10248.888,E2 -10248.888} C_VEL
LIN {X 0,Y 418.878,Z 729.305,A -85,B 0,C 180,E1 -10250.097,E2 -10250.097} C_VEL
LIN {X 0,Y 418.195,Z 737.193,A -85,B 0,C 180,E1 -10251.544,E2 -10251.544} C_VEL
LIN {X 0,Y 417.858,Z 743.143,A -85,B 0,C 180,E1 -10252.9,E2 -10252.9} C_VEL
LIN {X 0,Y 417.549,Z 747.792,A -85,B 0,C 180,E1 -10254.204,E2 -10254.204} C_VEL
LIN {X 0,Y 417.415,Z 751.825,A -85,B 0,C 180,E1 -10255.655,E2 -10255.655} C_VEL
LIN {X 0,Y 417.249,Z 754.793,A -85,B 0,C 180,E1 -10257.104,E2 -10257.104} C_VEL
LIN {X 0,Y 417.11,Z 756.193,A -85,B 0,C 180,E1 -10258.069,E2 -10258.069} C_VEL
LIN {X 0,Y 417.038,Z 757.176,A -85,B 0,C 180,E1 -10259.034,E2 -10259.034} C_VEL
LIN {X 0,Y 417.005,Z 757.749,A -85,B 0,C 180,E1 -10260,E2 -10260} C_VEL
LIN {X 0,Y 417.014,Z 757.883,A -85,B 0,C 180,E1 -10260.966,E2 -10260.966} C_VEL
LIN {X 0,Y 417.078,Z 757.571,A -85,B 0,C 180,E1 -10261.931,E2 -10261.931} C_VEL
LIN {X 0,Y 417.103,Z 756.852,A -85,B 0,C 180,E1 -10262.897,E2 -10262.897} C_VEL
LIN {X 0,Y 417.065,Z 755.725,A -85,B 0,C 180,E1 -10263.865,E2 -10263.865} C_VEL
LIN {X 0,Y 417.184,Z 753.172,A -85,B 0,C 180,E1 -10265.316,E2 -10265.316} C_VEL
LIN {X 0,Y 417.282,Z 749.294,A -85,B 0,C 180,E1 -10266.865,E2 -10266.865} C_VEL
LIN {X 0,Y 417.5,Z 744.846,A -85,B 0,C 180,E1 -10268.226,E2 -10268.226} C_VEL
LIN {X 0,Y 417.792,Z 738.826,A -85,B 0,C 180,E1 -10269.684,E2 -10269.684} C_VEL
LIN {X 0,Y 418.206,Z 731.287,A -85,B 0,C 180,E1 -10271.143,E2 -10271.143} C_VEL
LIN {X 0,Y 418.839,Z 721.938,A -85,B 0,C 180,E1 -10272.6,E2 -10272.6} C_VEL
LIN {X 0,Y 419.284,Z 713.353,A -85,B 0,C 180,E1 -10273.695,E2 -10273.695} C_VEL
LIN {X 0,Y 419.911,Z 702.912,A -85,B 0,C 180,E1 -10274.788,E2 -10274.788} C_VEL
LIN {X 0,Y 420.617,Z 691.423,A -85,B 0,C 180,E1 -10275.755,E2 -10275.755} C_VEL
LIN {X 0,Y 421.208,Z 679.655,A -85,B 0,C 180,E1 -10276.541,E2 -10276.541} C_VEL
LIN {X 0,Y 421.67,Z 666.341,A -85,B 0,C 180,E1 -10277.208,E2 -10277.208} C_VEL
LIN {X 0,Y 422.195,Z 652.417,A -85,B 0,C 180,E1 -10277.686,E2 -10277.686} C_VEL
LIN {X 0,Y 423.94,Z 562.944,A -85,B 0,C 180,E1 -10279.552,E2 -10279.552} C_VEL
LIN {X 0,Y 420.46,Z 540.233,A -85,B 0,C 180,E1 -10280.23,E2 -10280.23} C_VEL
LIN {X 0,Y 421.827,Z 518.778,A -85,B 0,C 180,E1 -10284.091,E2 -10284.091} C_VEL
LIN {X 0,Y 422.847,Z 504.667,A -85,B 0,C 180,E1 -10286.664,E2 -10286.664} C_VEL
LIN {X 0,Y 420.474,Z 493.125,A -85,B 0,C 180,E1 -10288.994,E2 -10288.994} C_VEL
LIN {X 0,Y 418.242,Z 483.513,A -85,B 0,C 180,E1 -10291.019,E2 -10291.019} C_VEL
LIN {X 0,Y 418.251,Z 483.514,A -85,B 0,C 180,E1 -10293.677,E2 -10293.677} C_VEL
LIN {X 0,Y 418.248,Z 483.51,A -85,B 0,C 180,E1 -10297.223,E2 -10297.223} C_VEL
LIN {X 0,Y 418.258,Z 483.512,A -85,B 0,C 180,E1 -10299.681,E2 -10299.681} C_VEL
LIN {X 0,Y 418.232,Z 483.509,A -85,B 0,C 180,E1 -10302.321,E2 -10302.321} C_VEL
LIN {X 0,Y 418.237,Z 483.51,A -85,B 0,C 180,E1 -10305.108,E2 -10305.108} C_VEL
LIN {X 0,Y 418.242,Z 483.513,A -85,B 0,C 180,E1 -10307.767,E2 -10307.767} C_VEL
LIN {X 0,Y 418.247,Z 483.507,A -85,B 0,C 180,E1 -10310.62,E2 -10310.62} C_VEL
LIN {X 0,Y 418.245,Z 483.51,A -85,B 0,C 180,E1 -10313.976,E2 -10313.976} C_VEL
LIN {X 0,Y 418.259,Z 483.508,A -85,B 0,C 180,E1 -10317.156,E2 -10317.156} C_VEL
LIN {X 0,Y 418.27,Z 483.505,A -85,B 0,C 180,E1 -10320.895,E2 -10320.895} C_VEL
LIN {X 0,Y 418.272,Z 483.505,A -85,B 0,C 180,E1 -10324.096,E2 -10324.096} C_VEL
LIN {X 0,Y 418.24,Z 483.512,A -85,B 0,C 180,E1 -10327.264,E2 -10327.264} C_VEL
LIN {X 0,Y 418.285,Z 483.502,A -85,B 0,C 180,E1 -10330.364,E2 -10330.364} C_VEL
LIN {X 0,Y 418.319,Z 483.504,A -85,B 0,C 180,E1 -10333.405,E2 -10333.405} C_VEL
LIN {X 0,Y 418.348,Z 483.496,A -85,B 0,C 180,E1 -10336.999,E2 -10336.999} C_VEL
LIN {X 0,Y 418.344,Z 483.495,A -85,B 0,C 180,E1 -10340.329,E2 -10340.329} C_VEL
LIN {X 0,Y 418.496,Z 483.481,A -85,B 0,C 180,E1 -10343.249,E2 -10343.249} C_VEL
LIN {X 0,Y 418.478,Z 483.478,A -85,B 0,C 180,E1 -10344.379,E2 -10344.379} C_VEL
LIN {X 0,Y 417.71,Z 483.58,A -85,B 0,C 180,E1 -10345.182,E2 -10345.182} C_VEL
LIN {X 0,Y 414.884,Z 483.926,A -85,B 0,C 180,E1 -10346.489,E2 -10346.489} C_VEL
LIN {X 0,Y 412.557,Z 484.222,A -85,B 0,C 180,E1 -10347.545,E2 -10347.545} C_VEL
LIN {X 0,Y 411.557,Z 484.341,A -85,B 0,C 180,E1 -10348.36,E2 -10348.36} C_VEL
LIN {X 0,Y 411.471,Z 484.351,A -85,B 0,C 180,E1 -10348.635,E2 -10348.635} C_VEL
LIN {X 0,Y 411.644,Z 484.331,A -85,B 0,C 180,E1 -10350,E2 -10350} C_VEL
LIN {X 0,Y 411.468,Z 484.353,A -85,B 0,C 180,E1 -10352.937,E2 -10352.937} C_VEL
LIN {X 0,Y 411.46,Z 484.354,A -85,B 0,C 180,E1 -10356.867,E2 -10356.867} C_VEL
LIN {X 0,Y 411.356,Z 484.367,A -85,B 0,C 180,E1 -10358.845,E2 -10358.845} C_VEL
LIN {X 0,Y 411.286,Z 484.377,A -85,B 0,C 180,E1 -10361.833,E2 -10361.833} C_VEL
LIN {X 0,Y 411.263,Z 484.379,A -85,B 0,C 180,E1 -10364.853,E2 -10364.853} C_VEL
LIN {X 0,Y 411.254,Z 484.38,A -85,B 0,C 180,E1 -10367.915,E2 -10367.915} C_VEL
LIN {X 0,Y 411.198,Z 484.388,A -85,B 0,C 180,E1 -10371.034,E2 -10371.034} C_VEL
LIN {X 0,Y 411.228,Z 484.382,A -85,B 0,C 180,E1 -10374.215,E2 -10374.215} C_VEL
LIN {X 0,Y 411.26,Z 484.383,A -85,B 0,C 180,E1 -10377.478,E2 -10377.478} C_VEL
LIN {X 0,Y 411.191,Z 484.388,A -85,B 0,C 180,E1 -10380.848,E2 -10380.848} C_VEL
LIN {X 0,Y 411.207,Z 484.384,A -85,B 0,C 180,E1 -10384.334,E2 -10384.334} C_VEL
LIN {X 0,Y 411.198,Z 484.386,A -85,B 0,C 180,E1 -10387.974,E2 -10387.974} C_VEL
LIN {X 0,Y 411.185,Z 484.387,A -85,B 0,C 180,E1 -10390.504,E2 -10390.504} C_VEL
LIN {X 0,Y 411.179,Z 484.393,A -85,B 0,C 180,E1 -10393.133,E2 -10393.133} C_VEL
LIN {X 0,Y 411.17,Z 484.39,A -85,B 0,C 180,E1 -10395.881,E2 -10395.881} C_VEL
LIN {X 0,Y 411.165,Z 484.391,A -85,B 0,C 180,E1 -10398.772,E2 -10398.772} C_VEL
LIN {X 0,Y 411.196,Z 484.386,A -85,B 0,C 180,E1 -10402.026,E2 -10402.026} C_VEL
LIN {X 0,Y 411.208,Z 484.389,A -85,B 0,C 180,E1 -10405.667,E2 -10405.667} C_VEL
LIN {X 0,Y 411.191,Z 484.391,A -85,B 0,C 180,E1 -10409.153,E2 -10409.153} C_VEL
LIN {X 0,Y 411.222,Z 484.395,A -85,B 0,C 180,E1 -10410.573,E2 -10410.573} C_VEL
LIN {X 0,Y 414.622,Z 499.75,A -85,B 0,C 180,E1 -10413.309,E2 -10413.309} C_VEL
LIN {X 0,Y 415.527,Z 504.739,A -85,B 0,C 180,E1 -10414.182,E2 -10414.182} C_VEL
LIN {X 0,Y 414.73,Z 522.536,A -85,B 0,C 180,E1 -10417.061,E2 -10417.061} C_VEL
LIN {X 0,Y 413.84,Z 541.644,A -85,B 0,C 180,E1 -10420.145,E2 -10420.145} C_VEL
LIN {X 0,Y 413.614,Z 547.095,A -85,B 0,C 180,E1 -10421.02,E2 -10421.02} C_VEL
LIN {X 0,Y 416.527,Z 566.982,A -85,B 0,C 180,E1 -10421.572,E2 -10421.572} C_VEL
LIN {X 0,Y 414.91,Z 657.648,A -85,B 0,C 180,E1 -10423.454,E2 -10423.454} C_VEL
LIN {X 0,Y 414.467,Z 670.102,A -85,B 0,C 180,E1 -10423.879,E2 -10423.879} C_VEL
LIN {X 0,Y 413.917,Z 683.474,A -85,B 0,C 180,E1 -10424.552,E2 -10424.552} C_VEL
LIN {X 0,Y 413.366,Z 695.44,A -85,B 0,C 180,E1 -10425.355,E2 -10425.355} C_VEL
LIN {X 0,Y 412.792,Z 706.777,A -85,B 0,C 180,E1 -10426.336,E2 -10426.336} C_VEL
LIN {X 0,Y 412.126,Z 718.159,A -85,B 0,C 180,E1 -10427.567,E2 -10427.567} C_VEL
LIN {X 0,Y 411.494,Z 728.107,A -85,B 0,C 180,E1 -10428.922,E2 -10428.922} C_VEL
LIN {X 0,Y 410.942,Z 736.875,A -85,B 0,C 180,E1 -10430.401,E2 -10430.401} C_VEL
LIN {X 0,Y 410.545,Z 743.839,A -85,B 0,C 180,E1 -10431.881,E2 -10431.881} C_VEL
LIN {X 0,Y 410.321,Z 749.625,A -85,B 0,C 180,E1 -10433.429,E2 -10433.429} C_VEL
LIN {X 0,Y 410.143,Z 754.353,A -85,B 0,C 180,E1 -10435.085,E2 -10435.085} C_VEL
LIN {X 0,Y 410.014,Z 756.465,A -85,B 0,C 180,E1 -10436.069,E2 -10436.069} C_VEL
LIN {X 0,Y 410.001,Z 758.14,A -85,B 0,C 180,E1 -10437.052,E2 -10437.052} C_VEL
LIN {X 0,Y 410.008,Z 759.386,A -85,B 0,C 180,E1 -10438.035,E2 -10438.035} C_VEL
LIN {X 0,Y 409.939,Z 760.161,A -85,B 0,C 180,E1 -10439.018,E2 -10439.018} C_VEL
LIN {X 0,Y 409.926,Z 760.528,A -85,B 0,C 180,E1 -10440,E2 -10440} C_VEL
LIN {X 0,Y 409.939,Z 760.488,A -85,B 0,C 180,E1 -10440.982,E2 -10440.982} C_VEL
LIN {X 0,Y 410.013,Z 759.985,A -85,B 0,C 180,E1 -10441.965,E2 -10441.965} C_VEL
LIN {X 0,Y 410.085,Z 759.059,A -85,B 0,C 180,E1 -10442.947,E2 -10442.947} C_VEL
LIN {X 0,Y 410.043,Z 757.728,A -85,B 0,C 180,E1 -10443.931,E2 -10443.931} C_VEL
LIN {X 0,Y 410.271,Z 754.853,A -85,B 0,C 180,E1 -10445.406,E2 -10445.406} C_VEL
LIN {X 0,Y 410.491,Z 750.902,A -85,B 0,C 180,E1 -10446.883,E2 -10446.883} C_VEL
LIN {X 0,Y 410.826,Z 744.733,A -85,B 0,C 180,E1 -10448.609,E2 -10448.609} C_VEL
LIN {X 0,Y 411.328,Z 737.961,A -85,B 0,C 180,E1 -10450.086,E2 -10450.086} C_VEL
LIN {X 0,Y 411.948,Z 729.516,A -85,B 0,C 180,E1 -10451.564,E2 -10451.564} C_VEL
LIN {X 0,Y 412.603,Z 720.857,A -85,B 0,C 180,E1 -10452.793,E2 -10452.793} C_VEL
LIN {X 0,Y 413.357,Z 710.965,A -85,B 0,C 180,E1 -10453.942,E2 -10453.942} C_VEL
LIN {X 0,Y 414.004,Z 701.108,A -85,B 0,C 180,E1 -10454.878,E2 -10454.878} C_VEL
LIN {X 0,Y 414.561,Z 689.844,A -85,B 0,C 180,E1 -10455.738,E2 -10455.738} C_VEL
LIN {X 0,Y 415.323,Z 677.393,A -85,B 0,C 180,E1 -10456.466,E2 -10456.466} C_VEL
LIN {X 0,Y 415.862,Z 664.486,A -85,B 0,C 180,E1 -10457.012,E2 -10457.012} C_VEL
LIN {X 0,Y 416.271,Z 650.181,A -85,B 0,C 180,E1 -10457.407,E2 -10457.407} C_VEL
LIN {X 0,Y 418.532,Z 568.01,A -85,B 0,C 180,E1 -10459.279,E2 -10459.279} C_VEL
LIN {X 0,Y 416.472,Z 554.658,A -85,B 0,C 180,E1 -10459.769,E2 -10459.769} C_VEL
LIN {X 0,Y 415.21,Z 548.532,A -85,B 0,C 180,E1 -10460.045,E2 -10460.045} C_VEL
LIN {X 0,Y 416.414,Z 526.182,A -85,B 0,C 180,E1 -10463.631,E2 -10463.631} C_VEL
LIN {X 0,Y 417.417,Z 508.603,A -85,B 0,C 180,E1 -10466.463,E2 -10466.463} C_VEL
LIN {X 0,Y 415.823,Z 499.973,A -85,B 0,C 180,E1 -10468.033,E2 -10468.033} C_VEL
LIN {X 0,Y 413.261,Z 490.819,A -85,B 0,C 180,E1 -10469.851,E2 -10469.851} C_VEL
LIN {X 0,Y 411.194,Z 484.394,A -85,B 0,C 180,E1 -10471.233,E2 -10471.233} C_VEL
LIN {X 0,Y 411.208,Z 484.391,A -85,B 0,C 180,E1 -10474.333,E2 -10474.333} C_VEL
LIN {X 0,Y 411.198,Z 484.39,A -85,B 0,C 180,E1 -10477.973,E2 -10477.973} C_VEL
LIN {X 0,Y 411.184,Z 484.391,A -85,B 0,C 180,E1 -10480.504,E2 -10480.504} C_VEL
LIN {X 0,Y 411.175,Z 484.391,A -85,B 0,C 180,E1 -10483.133,E2 -10483.133} C_VEL
LIN {X 0,Y 411.175,Z 484.39,A -85,B 0,C 180,E1 -10485.88,E2 -10485.88} C_VEL
LIN {X 0,Y 411.199,Z 484.388,A -85,B 0,C 180,E1 -10488.766,E2 -10488.766} C_VEL
LIN {X 0,Y 411.203,Z 484.39,A -85,B 0,C 180,E1 -10492.027,E2 -10492.027} C_VEL
LIN {X 0,Y 411.208,Z 484.389,A -85,B 0,C 180,E1 -10495.667,E2 -10495.667} C_VEL
LIN {X 0,Y 411.205,Z 484.39,A -85,B 0,C 180,E1 -10499.154,E2 -10499.154} C_VEL
LIN {X 0,Y 411.257,Z 484.493,A -85,B 0,C 180,E1 -10499.939,E2 -10499.939} C_VEL
LIN {X 0,Y 415.223,Z 500.807,A -85,B 0,C 180,E1 -10503.037,E2 -10503.037} C_VEL
LIN {X 0,Y 416.86,Z 509.092,A -85,B 0,C 180,E1 -10504.538,E2 -10504.538} C_VEL
LIN {X 0,Y 415.464,Z 526.181,A -85,B 0,C 180,E1 -10507.267,E2 -10507.267} C_VEL
LIN {X 0,Y 418.903,Z 548.764,A -85,B 0,C 180,E1 -10507.905,E2 -10507.905} C_VEL
LIN {X 0,Y 416.625,Z 662.446,A -85,B 0,C 180,E1 -10510.187,E2 -10510.187} C_VEL
LIN {X 0,Y 416.021,Z 676.928,A -85,B 0,C 180,E1 -10510.67,E2 -10510.67} C_VEL
LIN {X 0,Y 415.425,Z 690.675,A -85,B 0,C 180,E1 -10511.332,E2 -10511.332} C_VEL
LIN {X 0,Y 414.719,Z 703.398,A -85,B 0,C 180,E1 -10512.134,E2 -10512.134} C_VEL
LIN {X 0,Y 413.901,Z 715.534,A -85,B 0,C 180,E1 -10513.095,E2 -10513.095} C_VEL
LIN {X 0,Y 413.053,Z 726.931,A -85,B 0,C 180,E1 -10514.203,E2 -10514.203} C_VEL
LIN {X 0,Y 412.278,Z 737.408,A -85,B 0,C 180,E1 -10515.437,E2 -10515.437} C_VEL
LIN {X 0,Y 411.588,Z 747.462,A -85,B 0,C 180,E1 -10516.874,E2 -10516.874} C_VEL
LIN {X 0,Y 411.076,Z 756.315,A -85,B 0,C 180,E1 -10518.411,E2 -10518.411} C_VEL
LIN {X 0,Y 410.545,Z 764.432,A -85,B 0,C 180,E1 -10520.143,E2 -10520.143} C_VEL
LIN {X 0,Y 410.258,Z 770.085,A -85,B 0,C 180,E1 -10521.627,E2 -10521.627} C_VEL
LIN {X 0,Y 410.085,Z 774.687,A -85,B 0,C 180,E1 -10523.11,E2 -10523.11} C_VEL
LIN {X 0,Y 409.995,Z 779.264,A -85,B 0,C 180,E1 -10525.083,E2 -10525.083} C_VEL
LIN {X 0,Y 409.927,Z 782.287,A -85,B 0,C 180,E1 -10527.052,E2 -10527.052} C_VEL
LIN {X 0,Y 409.994,Z 783.248,A -85,B 0,C 180,E1 -10528.035,E2 -10528.035} C_VEL
LIN {X 0,Y 409.925,Z 784.078,A -85,B 0,C 180,E1 -10530,E2 -10530} C_VEL
LIN {X 0,Y 409.976,Z 783.47,A -85,B 0,C 180,E1 -10531.965,E2 -10531.965} C_VEL
LIN {X 0,Y 409.922,Z 781.392,A -85,B 0,C 180,E1 -10533.932,E2 -10533.932} C_VEL
LIN {X 0,Y 410.035,Z 777.807,A -85,B 0,C 180,E1 -10535.903,E2 -10535.903} C_VEL
LIN {X 0,Y 410.155,Z 774.115,A -85,B 0,C 180,E1 -10537.384,E2 -10537.384} C_VEL
LIN {X 0,Y 410.362,Z 769.406,A -85,B 0,C 180,E1 -10538.867,E2 -10538.867} C_VEL
LIN {X 0,Y 410.746,Z 762.603,A -85,B 0,C 180,E1 -10540.599,E2 -10540.599} C_VEL
LIN {X 0,Y 411.387,Z 754.109,A -85,B 0,C 180,E1 -10542.33,E2 -10542.33} C_VEL
LIN {X 0,Y 412.049,Z 745.188,A -85,B 0,C 180,E1 -10543.815,E2 -10543.815} C_VEL
LIN {X 0,Y 412.839,Z 734.377,A -85,B 0,C 180,E1 -10545.3,E2 -10545.3} C_VEL
LIN {X 0,Y 413.79,Z 723.455,A -85,B 0,C 180,E1 -10546.529,E2 -10546.529} C_VEL
LIN {X 0,Y 414.72,Z 711.528,A -85,B 0,C 180,E1 -10547.633,E2 -10547.633} C_VEL
LIN {X 0,Y 415.672,Z 699.231,A -85,B 0,C 180,E1 -10548.552,E2 -10548.552} C_VEL
LIN {X 0,Y 416.527,Z 685.908,A -85,B 0,C 180,E1 -10549.337,E2 -10549.337} C_VEL
LIN {X 0,Y 417.215,Z 672.887,A -85,B 0,C 180,E1 -10549.913,E2 -10549.913} C_VEL
LIN {X 0,Y 417.823,Z 657.973,A -85,B 0,C 180,E1 -10550.364,E2 -10550.364} C_VEL
LIN {X 0,Y 420.139,Z 570.931,A -85,B 0,C 180,E1 -10552.235,E2 -10552.235} C_VEL
LIN {X 0,Y 420.737,Z 548.753,A -85,B 0,C 180,E1 -10552.746,E2 -10552.746} C_VEL
LIN {X 0,Y 418.803,Z 535.785,A -85,B 0,C 180,E1 -10553.223,E2 -10553.223} C_VEL
LIN {X 0,Y 417.153,Z 527.452,A -85,B 0,C 180,E1 -10553.597,E2 -10553.597} C_VEL
LIN {X 0,Y 418.974,Z 513.572,A -85,B 0,C 180,E1 -10556.112,E2 -10556.112} C_VEL
LIN {X 0,Y 417.297,Z 504.751,A -85,B 0,C 180,E1 -10558.136,E2 -10558.136} C_VEL
LIN {X 0,Y 414.748,Z 495.616,A -85,B 0,C 180,E1 -10560.555,E2 -10560.555} C_VEL
LIN {X 0,Y 412.203,Z 487.524,A -85,B 0,C 180,E1 -10563.066,E2 -10563.066} C_VEL
LIN {X 0,Y 411.211,Z 484.39,A -85,B 0,C 180,E1 -10564.185,E2 -10564.185} C_VEL
LIN {X 0,Y 411.192,Z 484.392,A -85,B 0,C 180,E1 -10566.742,E2 -10566.742} C_VEL
LIN {X 0,Y 411.217,Z 484.388,A -85,B 0,C 180,E1 -10569.728,E2 -10569.728} C_VEL
LIN {X 0,Y 411.18,Z 484.393,A -85,B 0,C 180,E1 -10573.133,E2 -10573.133} C_VEL
LIN {X 0,Y 411.171,Z 484.393,A -85,B 0,C 180,E1 -10575.881,E2 -10575.881} C_VEL
LIN {X 0,Y 411.167,Z 484.395,A -85,B 0,C 180,E1 -10578.772,E2 -10578.772} C_VEL
LIN {X 0,Y 411.209,Z 484.39,A -85,B 0,C 180,E1 -10581.831,E2 -10581.831} C_VEL
LIN {X 0,Y 411.214,Z 484.39,A -85,B 0,C 180,E1 -10585.122,E2 -10585.122} C_VEL
LIN {X 0,Y 411.216,Z 484.51,A -85,B 0,C 180,E1 -10586.699,E2 -10586.699} C_VEL
LIN {X 0,Y 413.628,Z 492.132,A -85,B 0,C 180,E1 -10589.354,E2 -10589.354} C_VEL
LIN {X 0,Y 415.938,Z 500.182,A -85,B 0,C 180,E1 -10591.764,E2 -10591.764} C_VEL
LIN {X 0,Y 417.718,Z 509.016,A -85,B 0,C 180,E1 -10594.059,E2 -10594.059} C_VEL
LIN {X 0,Y 418.079,Z 512.487,A -85,B 0,C 180,E1 -10594.884,E2 -10594.884} C_VEL
LIN {X 0,Y 415.897,Z 530.619,A -85,B 0,C 180,E1 -10598.554,E2 -10598.554} C_VEL
LIN {X 0,Y 415.104,Z 539.56,A -85,B 0,C 180,E1 -10600.265,E2 -10600.265} C_VEL
LIN {X 0,Y 418.736,Z 557.74,A -85,B 0,C 180,E1 -10601.072,E2 -10601.072} C_VEL
LIN {X 0,Y 419.779,Z 565.866,A -85,B 0,C 180,E1 -10601.382,E2 -10601.382} C_VEL
LIN {X 0,Y 417.048,Z 645.047,A -85,B 0,C 180,E1 -10603.321,E2 -10603.321} C_VEL
LIN {X 0,Y 416.49,Z 659.54,A -85,B 0,C 180,E1 -10603.739,E2 -10603.739} C_VEL
LIN {X 0,Y 415.804,Z 674.073,A -85,B 0,C 180,E1 -10604.386,E2 -10604.386} C_VEL
LIN {X 0,Y 415.081,Z 687.165,A -85,B 0,C 180,E1 -10605.19,E2 -10605.19} C_VEL
LIN {X 0,Y 414.265,Z 699.149,A -85,B 0,C 180,E1 -10606.135,E2 -10606.135} C_VEL
LIN {X 0,Y 413.266,Z 710.261,A -85,B 0,C 180,E1 -10607.228,E2 -10607.228} C_VEL
LIN {X 0,Y 412.583,Z 720.218,A -85,B 0,C 180,E1 -10608.454,E2 -10608.454} C_VEL
LIN {X 0,Y 411.93,Z 729.936,A -85,B 0,C 180,E1 -10609.928,E2 -10609.928} C_VEL
LIN {X 0,Y 411.203,Z 737.718,A -85,B 0,C 180,E1 -10611.399,E2 -10611.399} C_VEL
LIN {X 0,Y 410.809,Z 743.949,A -85,B 0,C 180,E1 -10612.864,E2 -10612.864} C_VEL
LIN {X 0,Y 410.518,Z 748.234,A -85,B 0,C 180,E1 -10614.104,E2 -10614.104} C_VEL
LIN {X 0,Y 410.35,Z 752.227,A -85,B 0,C 180,E1 -10615.58,E2 -10615.58} C_VEL
LIN {X 0,Y 410.189,Z 755.151,A -85,B 0,C 180,E1 -10617.054,E2 -10617.054} C_VEL
LIN {X 0,Y 410.041,Z 756.521,A -85,B 0,C 180,E1 -10618.036,E2 -10618.036} C_VEL
LIN {X 0,Y 409.962,Z 757.476,A -85,B 0,C 180,E1 -10619.018,E2 -10619.018} C_VEL
LIN {X 0,Y 409.927,Z 758.021,A -85,B 0,C 180,E1 -10620,E2 -10620} C_VEL
LIN {X 0,Y 409.939,Z 758.105,A -85,B 0,C 180,E1 -10620.982,E2 -10620.982} C_VEL
LIN {X 0,Y 410.008,Z 757.764,A -85,B 0,C 180,E1 -10621.965,E2 -10621.965} C_VEL
LIN {X 0,Y 410.002,Z 757.019,A -85,B 0,C 180,E1 -10622.948,E2 -10622.948} C_VEL
LIN {X 0,Y 409.981,Z 755.856,A -85,B 0,C 180,E1 -10623.932,E2 -10623.932} C_VEL
LIN {X 0,Y 410.111,Z 753.247,A -85,B 0,C 180,E1 -10625.408,E2 -10625.408} C_VEL
LIN {X 0,Y 410.193,Z 749.585,A -85,B 0,C 180,E1 -10626.888,E2 -10626.888} C_VEL
LIN {X 0,Y 410.441,Z 744.77,A -85,B 0,C 180,E1 -10628.369,E2 -10628.369} C_VEL
LIN {X 0,Y 410.768,Z 738.646,A -85,B 0,C 180,E1 -10629.851,E2 -10629.851} C_VEL
LIN {X 0,Y 411.217,Z 731.002,A -85,B 0,C 180,E1 -10631.335,E2 -10631.335} C_VEL
LIN {X 0,Y 411.738,Z 723.234,A -85,B 0,C 180,E1 -10632.57,E2 -10632.57} C_VEL
LIN {X 0,Y 412.252,Z 713.842,A -85,B 0,C 180,E1 -10633.808,E2 -10633.808} C_VEL
LIN {X 0,Y 412.9,Z 703.491,A -85,B 0,C 180,E1 -10634.918,E2 -10634.918} C_VEL
LIN {X 0,Y 413.639,Z 692.09,A -85,B 0,C 180,E1 -10635.901,E2 -10635.901} C_VEL
LIN {X 0,Y 414.311,Z 679.469,A -85,B 0,C 180,E1 -10636.761,E2 -10636.761} C_VEL
LIN {X 0,Y 414.751,Z 666.036,A -85,B 0,C 180,E1 -10637.441,E2 -10637.441} C_VEL
LIN {X 0,Y 415.32,Z 652.014,A -85,B 0,C 180,E1 -10637.925,E2 -10637.925} C_VEL
LIN {X 0,Y 417.134,Z 563.669,A -85,B 0,C 180,E1 -10639.814,E2 -10639.814} C_VEL
LIN {X 0,Y 413.528,Z 540.216,A -85,B 0,C 180,E1 -10640.518,E2 -10640.518} C_VEL
LIN {X 0,Y 414.918,Z 519.782,A -85,B 0,C 180,E1 -10644.252,E2 -10644.252} C_VEL
LIN {X 0,Y 415.927,Z 506.827,A -85,B 0,C 180,E1 -10646.649,E2 -10646.649} C_VEL
LIN {X 0,Y 414.784,Z 500.108,A -85,B 0,C 180,E1 -10647.999,E2 -10647.999} C_VEL
LIN {X 0,Y 411.191,Z 484.393,A -85,B 0,C 180,E1 -10651.316,E2 -10651.316} C_VEL
LIN {X 0,Y 411.209,Z 484.388,A -85,B 0,C 180,E1 -10654.333,E2 -10654.333} C_VEL
LIN {X 0,Y 411.203,Z 484.388,A -85,B 0,C 180,E1 -10657.973,E2 -10657.973} C_VEL
LIN {X 0,Y 411.186,Z 484.387,A -85,B 0,C 180,E1 -10660.504,E2 -10660.504} C_VEL
LIN {X 0,Y 411.176,Z 484.39,A -85,B 0,C 180,E1 -10663.133,E2 -10663.133} C_VEL
LIN {X 0,Y 411.169,Z 484.392,A -85,B 0,C 180,E1 -10665.881,E2 -10665.881} C_VEL
LIN {X 0,Y 411.165,Z 484.39,A -85,B 0,C 180,E1 -10668.772,E2 -10668.772} C_VEL
LIN {X 0,Y 411.193,Z 484.388,A -85,B 0,C 180,E1 -10672.026,E2 -10672.026} C_VEL
LIN {X 0,Y 411.208,Z 484.39,A -85,B 0,C 180,E1 -10675.666,E2 -10675.666} C_VEL
LIN {X 0,Y 411.191,Z 484.389,A -85,B 0,C 180,E1 -10679.152,E2 -10679.152} C_VEL
LIN {X 0,Y 411.26,Z 484.377,A -85,B 0,C 180,E1 -10682.522,E2 -10682.522} C_VEL
LIN {X 0,Y 411.229,Z 484.385,A -85,B 0,C 180,E1 -10685.785,E2 -10685.785} C_VEL
LIN {X 0,Y 411.198,Z 484.387,A -85,B 0,C 180,E1 -10688.966,E2 -10688.966} C_VEL
LIN {X 0,Y 411.255,Z 484.379,A -85,B 0,C 180,E1 -10692.085,E2 -10692.085} C_VEL
LIN {X 0,Y 411.263,Z 484.38,A -85,B 0,C 180,E1 -10695.147,E2 -10695.147} C_VEL
LIN {X 0,Y 411.286,Z 484.375,A -85,B 0,C 180,E1 -10698.167,E2 -10698.167} C_VEL
LIN {X 0,Y 411.483,Z 484.35,A -85,B 0,C 180,E1 -10702.147,E2 -10702.147} C_VEL
LIN {X 0,Y 411.427,Z 484.357,A -85,B 0,C 180,E1 -10704.351,E2 -10704.351} C_VEL
LIN {X 0,Y 411.516,Z 484.347,A -85,B 0,C 180,E1 -10708.043,E2 -10708.043} C_VEL
LIN {X 0,Y 411.471,Z 484.351,A -85,B 0,C 180,E1 -10708.635,E2 -10708.635} C_VEL
LIN {X 0,Y 410.789,Z 484.444,A -85,B 0,C 180,E1 -10709.452,E2 -10709.452} C_VEL
LIN {X 0,Y 407.935,Z 484.792,A -85,B 0,C 180,E1 -10710.779,E2 -10710.779} C_VEL
LIN {X 0,Y 405.533,Z 485.094,A -85,B 0,C 180,E1 -10711.852,E2 -10711.852} C_VEL
LIN {X 0,Y 404.506,Z 485.22,A -85,B 0,C 180,E1 -10712.68,E2 -10712.68} C_VEL
LIN {X 0,Y 404.425,Z 485.231,A -85,B 0,C 180,E1 -10712.961,E2 -10712.961} C_VEL
LIN {X 0,Y 404.412,Z 485.233,A -85,B 0,C 180,E1 -10716.987,E2 -10716.987} C_VEL
LIN {X 0,Y 404.26,Z 485.251,A -85,B 0,C 180,E1 -10720.012,E2 -10720.012} C_VEL
LIN {X 0,Y 404.268,Z 485.253,A -85,B 0,C 180,E1 -10723.211,E2 -10723.211} C_VEL
LIN {X 0,Y 404.217,Z 485.258,A -85,B 0,C 180,E1 -10727.007,E2 -10727.007} C_VEL
LIN {X 0,Y 404.165,Z 485.261,A -85,B 0,C 180,E1 -10730.352,E2 -10730.352} C_VEL
LIN {X 0,Y 404.171,Z 485.265,A -85,B 0,C 180,E1 -10733.574,E2 -10733.574} C_VEL
LIN {X 0,Y 404.185,Z 485.261,A -85,B 0,C 180,E1 -10735.766,E2 -10735.766} C_VEL
LIN {X 0,Y 404.197,Z 485.258,A -85,B 0,C 180,E1 -10738,E2 -10738} C_VEL
LIN {X 0,Y 404.141,Z 485.269,A -85,B 0,C 180,E1 -10741.558,E2 -10741.558} C_VEL
LIN {X 0,Y 404.186,Z 485.262,A -85,B 0,C 180,E1 -10745.016,E2 -10745.016} C_VEL
LIN {X 0,Y 404.158,Z 485.263,A -85,B 0,C 180,E1 -10748.757,E2 -10748.757} C_VEL
LIN {X 0,Y 404.127,Z 485.27,A -85,B 0,C 180,E1 -10751.6,E2 -10751.6} C_VEL
LIN {X 0,Y 404.15,Z 485.263,A -85,B 0,C 180,E1 -10754.523,E2 -10754.523} C_VEL
LIN {X 0,Y 404.138,Z 485.272,A -85,B 0,C 180,E1 -10757.296,E2 -10757.296} C_VEL
LIN {X 0,Y 404.17,Z 485.261,A -85,B 0,C 180,E1 -10759.956,E2 -10759.956} C_VEL
LIN {X 0,Y 404.138,Z 485.27,A -85,B 0,C 180,E1 -10763.125,E2 -10763.125} C_VEL
LIN {X 0,Y 404.147,Z 485.264,A -85,B 0,C 180,E1 -10766.188,E2 -10766.188} C_VEL
LIN {X 0,Y 404.166,Z 485.264,A -85,B 0,C 180,E1 -10769.717,E2 -10769.717} C_VEL
LIN {X 0,Y 404.225,Z 485.362,A -85,B 0,C 180,E1 -10770.32,E2 -10770.32} C_VEL
LIN {X 0,Y 407.611,Z 500.701,A -85,B 0,C 180,E1 -10773.089,E2 -10773.089} C_VEL
LIN {X 0,Y 408.615,Z 505.982,A -85,B 0,C 180,E1 -10774.02,E2 -10774.02} C_VEL
LIN {X 0,Y 407.798,Z 523.666,A -85,B 0,C 180,E1 -10776.916,E2 -10776.916} C_VEL
LIN {X 0,Y 406.884,Z 542.946,A -85,B 0,C 180,E1 -10780.054,E2 -10780.054} C_VEL
LIN {X 0,Y 406.69,Z 547.195,A -85,B 0,C 180,E1 -10780.742,E2 -10780.742} C_VEL
LIN {X 0,Y 409.688,Z 568.21,A -85,B 0,C 180,E1 -10781.334,E2 -10781.334} C_VEL
LIN {X 0,Y 407.961,Z 658.168,A -85,B 0,C 180,E1 -10783.261,E2 -10783.261} C_VEL
LIN {X 0,Y 407.501,Z 671.135,A -85,B 0,C 180,E1 -10783.724,E2 -10783.724} C_VEL
LIN {X 0,Y 406.912,Z 684.248,A -85,B 0,C 180,E1 -10784.408,E2 -10784.408} C_VEL
LIN {X 0,Y 406.329,Z 696.318,A -85,B 0,C 180,E1 -10785.245,E2 -10785.245} C_VEL
LIN {X 0,Y 405.776,Z 707.313,A -85,B 0,C 180,E1 -10786.223,E2 -10786.223} C_VEL
LIN {X 0,Y 405.088,Z 718.631,A -85,B 0,C 180,E1 -10787.475,E2 -10787.475} C_VEL
LIN {X 0,Y 404.487,Z 727.719,A -85,B 0,C 180,E1 -10788.728,E2 -10788.728} C_VEL
LIN {X 0,Y 403.914,Z 736.607,A -85,B 0,C 180,E1 -10790.233,E2 -10790.233} C_VEL
LIN {X 0,Y 403.482,Z 743.685,A -85,B 0,C 180,E1 -10791.738,E2 -10791.738} C_VEL
LIN {X 0,Y 403.212,Z 750.069,A -85,B 0,C 180,E1 -10793.471,E2 -10793.471} C_VEL
LIN {X 0,Y 403.06,Z 754.353,A -85,B 0,C 180,E1 -10794.998,E2 -10794.998} C_VEL
LIN {X 0,Y 402.933,Z 756.517,A -85,B 0,C 180,E1 -10795.999,E2 -10795.999} C_VEL
LIN {X 0,Y 402.902,Z 758.22,A -85,B 0,C 180,E1 -10797,E2 -10797} C_VEL
LIN {X 0,Y 402.921,Z 759.508,A -85,B 0,C 180,E1 -10798.001,E2 -10798.001} C_VEL
LIN {X 0,Y 402.867,Z 760.326,A -85,B 0,C 180,E1 -10799,E2 -10799} C_VEL
LIN {X 0,Y 402.851,Z 760.718,A -85,B 0,C 180,E1 -10800,E2 -10800} C_VEL
LIN {X 0,Y 402.867,Z 760.704,A -85,B 0,C 180,E1 -10801,E2 -10801} C_VEL
LIN {X 0,Y 402.946,Z 760.241,A -85,B 0,C 180,E1 -10801.999,E2 -10801.999} C_VEL
LIN {X 0,Y 402.989,Z 759.334,A -85,B 0,C 180,E1 -10802.999,E2 -10802.999} C_VEL
LIN {X 0,Y 402.961,Z 758.019,A -85,B 0,C 180,E1 -10804,E2 -10804} C_VEL
LIN {X 0,Y 403.226,Z 755.174,A -85,B 0,C 180,E1 -10805.501,E2 -10805.501} C_VEL
LIN {X 0,Y 403.447,Z 751.254,A -85,B 0,C 180,E1 -10807.004,E2 -10807.004} C_VEL
LIN {X 0,Y 403.818,Z 745.159,A -85,B 0,C 180,E1 -10808.759,E2 -10808.759} C_VEL
LIN {X 0,Y 404.35,Z 738.458,A -85,B 0,C 180,E1 -10810.262,E2 -10810.262} C_VEL
LIN {X 0,Y 405.014,Z 730.091,A -85,B 0,C 180,E1 -10811.765,E2 -10811.765} C_VEL
LIN {X 0,Y 405.707,Z 721.477,A -85,B 0,C 180,E1 -10813.014,E2 -10813.014} C_VEL
LIN {X 0,Y 406.524,Z 711.671,A -85,B 0,C 180,E1 -10814.178,E2 -10814.178} C_VEL
LIN {X 0,Y 407.302,Z 700.428,A -85,B 0,C 180,E1 -10815.256,E2 -10815.256} C_VEL
LIN {X 0,Y 407.906,Z 689.059,A -85,B 0,C 180,E1 -10816.13,E2 -10816.13} C_VEL
LIN {X 0,Y 408.761,Z 676.389,A -85,B 0,C 180,E1 -10816.866,E2 -10816.866} C_VEL
LIN {X 0,Y 409.352,Z 662.233,A -85,B 0,C 180,E1 -10817.452,E2 -10817.452} C_VEL
LIN {X 0,Y 409.799,Z 645.323,A -85,B 0,C 180,E1 -10817.884,E2 -10817.884} C_VEL
LIN {X 0,Y 412.136,Z 569.303,A -85,B 0,C 180,E1 -10819.681,E2 -10819.681} C_VEL
LIN {X 0,Y 410.466,Z 557.626,A -85,B 0,C 180,E1 -10820.122,E2 -10820.122} C_VEL
LIN {X 0,Y 408.62,Z 548.844,A -85,B 0,C 180,E1 -10820.514,E2 -10820.514} C_VEL
LIN {X 0,Y 409.793,Z 528.837,A -85,B 0,C 180,E1 -10823.768,E2 -10823.768} C_VEL
LIN {X 0,Y 410.895,Z 511.472,A -85,B 0,C 180,E1 -10826.597,E2 -10826.597} C_VEL
LIN {X 0,Y 409.979,Z 505.039,A -85,B 0,C 180,E1 -10827.795,E2 -10827.795} C_VEL
LIN {X 0,Y 407.66,Z 495.988,A -85,B 0,C 180,E1 -10829.601,E2 -10829.601} C_VEL
LIN {X 0,Y 404.141,Z 485.273,A -85,B 0,C 180,E1 -10831.969,E2 -10831.969} C_VEL
LIN {X 0,Y 404.183,Z 485.266,A -85,B 0,C 180,E1 -10835.19,E2 -10835.19} C_VEL
LIN {X 0,Y 404.158,Z 485.266,A -85,B 0,C 180,E1 -10838.757,E2 -10838.757} C_VEL
LIN {X 0,Y 404.125,Z 485.269,A -85,B 0,C 180,E1 -10841.6,E2 -10841.6} C_VEL
LIN {X 0,Y 404.148,Z 485.27,A -85,B 0,C 180,E1 -10844.522,E2 -10844.522} C_VEL
LIN {X 0,Y 404.175,Z 485.262,A -85,B 0,C 180,E1 -10847.3,E2 -10847.3} C_VEL
LIN {X 0,Y 404.17,Z 485.265,A -85,B 0,C 180,E1 -10849.955,E2 -10849.955} C_VEL
LIN {X 0,Y 404.142,Z 485.268,A -85,B 0,C 180,E1 -10853.124,E2 -10853.124} C_VEL
LIN {X 0,Y 404.147,Z 485.267,A -85,B 0,C 180,E1 -10856.188,E2 -10856.188} C_VEL
LIN {X 0,Y 404.224,Z 485.429,A -85,B 0,C 180,E1 -10859.613,E2 -10859.613} C_VEL
LIN {X 0,Y 408.291,Z 502.216,A -85,B 0,C 180,E1 -10862.861,E2 -10862.861} C_VEL
LIN {X 0,Y 409.962,Z 510.251,A -85,B 0,C 180,E1 -10864.351,E2 -10864.351} C_VEL
LIN {X 0,Y 408.582,Z 526.084,A -85,B 0,C 180,E1 -10866.952,E2 -10866.952} C_VEL
LIN {X 0,Y 412.129,Z 549.974,A -85,B 0,C 180,E1 -10867.633,E2 -10867.633} C_VEL
LIN {X 0,Y 409.767,Z 662.165,A -85,B 0,C 180,E1 -10869.939,E2 -10869.939} C_VEL
LIN {X 0,Y 409.116,Z 676.64,A -85,B 0,C 180,E1 -10870.429,E2 -10870.429} C_VEL
LIN {X 0,Y 408.511,Z 690.801,A -85,B 0,C 180,E1 -10871.123,E2 -10871.123} C_VEL
LIN {X 0,Y 407.767,Z 703.294,A -85,B 0,C 180,E1 -10871.927,E2 -10871.927} C_VEL
LIN {X 0,Y 406.915,Z 715.677,A -85,B 0,C 180,E1 -10872.926,E2 -10872.926} C_VEL
LIN {X 0,Y 406.041,Z 727.029,A -85,B 0,C 180,E1 -10874.051,E2 -10874.051} C_VEL
LIN {X 0,Y 405.175,Z 738.384,A -85,B 0,C 180,E1 -10875.433,E2 -10875.433} C_VEL
LIN {X 0,Y 404.494,Z 748.55,A -85,B 0,C 180,E1 -10876.946,E2 -10876.946} C_VEL
LIN {X 0,Y 403.958,Z 756.942,A -85,B 0,C 180,E1 -10878.459,E2 -10878.459} C_VEL
LIN {X 0,Y 403.451,Z 764.92,A -85,B 0,C 180,E1 -10880.221,E2 -10880.221} C_VEL
LIN {X 0,Y 403.126,Z 771.273,A -85,B 0,C 180,E1 -10881.983,E2 -10881.983} C_VEL
LIN {X 0,Y 402.939,Z 776.393,A -85,B 0,C 180,E1 -10883.819,E2 -10883.819} C_VEL
LIN {X 0,Y 402.909,Z 778.912,A -85,B 0,C 180,E1 -10884.997,E2 -10884.997} C_VEL
LIN {X 0,Y 402.828,Z 781.983,A -85,B 0,C 180,E1 -10887,E2 -10887} C_VEL
LIN {X 0,Y 402.904,Z 782.966,A -85,B 0,C 180,E1 -10888.001,E2 -10888.001} C_VEL
LIN {X 0,Y 402.85,Z 783.834,A -85,B 0,C 180,E1 -10890,E2 -10890} C_VEL
LIN {X 0,Y 402.888,Z 783.258,A -85,B 0,C 180,E1 -10891.999,E2 -10891.999} C_VEL
LIN {X 0,Y 402.842,Z 781.222,A -85,B 0,C 180,E1 -10894.002,E2 -10894.002} C_VEL
LIN {X 0,Y 402.908,Z 779.635,A -85,B 0,C 180,E1 -10895.004,E2 -10895.004} C_VEL
LIN {X 0,Y 403.066,Z 775.293,A -85,B 0,C 180,E1 -10897.011,E2 -10897.011} C_VEL
LIN {X 0,Y 403.308,Z 769.298,A -85,B 0,C 180,E1 -10899.023,E2 -10899.023} C_VEL
LIN {X 0,Y 403.731,Z 762.516,A -85,B 0,C 180,E1 -10900.786,E2 -10900.786} C_VEL
LIN {X 0,Y 404.405,Z 754.074,A -85,B 0,C 180,E1 -10902.547,E2 -10902.547} C_VEL
LIN {X 0,Y 405.126,Z 745.196,A -85,B 0,C 180,E1 -10904.056,E2 -10904.056} C_VEL
LIN {X 0,Y 405.95,Z 734.431,A -85,B 0,C 180,E1 -10905.566,E2 -10905.566} C_VEL
LIN {X 0,Y 406.983,Z 723.58,A -85,B 0,C 180,E1 -10906.813,E2 -10906.813} C_VEL
LIN {X 0,Y 407.953,Z 711.735,A -85,B 0,C 180,E1 -10907.935,E2 -10907.935} C_VEL
LIN {X 0,Y 409.02,Z 698.848,A -85,B 0,C 180,E1 -10908.919,E2 -10908.919} C_VEL
LIN {X 0,Y 409.919,Z 685.285,A -85,B 0,C 180,E1 -10909.727,E2 -10909.727} C_VEL
LIN {X 0,Y 410.752,Z 671.327,A -85,B 0,C 180,E1 -10910.338,E2 -10910.338} C_VEL
LIN {X 0,Y 411.345,Z 655.884,A -85,B 0,C 180,E1 -10910.797,E2 -10910.797} C_VEL
LIN {X 0,Y 413.651,Z 575.752,A -85,B 0,C 180,E1 -10912.573,E2 -10912.573} C_VEL
LIN {X 0,Y 414.468,Z 549.59,A -85,B 0,C 180,E1 -10913.193,E2 -10913.193} C_VEL
LIN {X 0,Y 412.508,Z 536.433,A -85,B 0,C 180,E1 -10913.704,E2 -10913.704} C_VEL
LIN {X 0,Y 410.716,Z 527.794,A -85,B 0,C 180,E1 -10914.105,E2 -10914.105} C_VEL
LIN {X 0,Y 412.437,Z 515.99,A -85,B 0,C 180,E1 -10916.298,E2 -10916.298} C_VEL
LIN {X 0,Y 410.828,Z 507.337,A -85,B 0,C 180,E1 -10918.341,E2 -10918.341} C_VEL
LIN {X 0,Y 408.509,Z 498.862,A -85,B 0,C 180,E1 -10920.661,E2 -10920.661} C_VEL
LIN {X 0,Y 406.28,Z 491.629,A -85,B 0,C 180,E1 -10922.961,E2 -10922.961} C_VEL
LIN {X 0,Y 404.17,Z 485.268,A -85,B 0,C 180,E1 -10925.419,E2 -10925.419} C_VEL
LIN {X 0,Y 404.158,Z 485.268,A -85,B 0,C 180,E1 -10928.757,E2 -10928.757} C_VEL
LIN {X 0,Y 404.127,Z 485.273,A -85,B 0,C 180,E1 -10931.6,E2 -10931.6} C_VEL
LIN {X 0,Y 404.151,Z 485.267,A -85,B 0,C 180,E1 -10934.523,E2 -10934.523} C_VEL
LIN {X 0,Y 404.139,Z 485.271,A -85,B 0,C 180,E1 -10937.296,E2 -10937.296} C_VEL
LIN {X 0,Y 404.171,Z 485.266,A -85,B 0,C 180,E1 -10939.956,E2 -10939.956} C_VEL
LIN {X 0,Y 404.139,Z 485.271,A -85,B 0,C 180,E1 -10943.125,E2 -10943.125} C_VEL
LIN {X 0,Y 404.192,Z 485.454,A -85,B 0,C 180,E1 -10945.515,E2 -10945.515} C_VEL
LIN {X 0,Y 406.541,Z 492.711,A -85,B 0,C 180,E1 -10948.344,E2 -10948.344} C_VEL
LIN {X 0,Y 408.596,Z 499.75,A -85,B 0,C 180,E1 -10950.646,E2 -10950.646} C_VEL
LIN {X 0,Y 410.152,Z 505.965,A -85,B 0,C 180,E1 -10952.442,E2 -10952.442} C_VEL
LIN {X 0,Y 411.518,Z 513.736,A -85,B 0,C 180,E1 -10954.455,E2 -10954.455} C_VEL
LIN {X 0,Y 410.237,Z 523.53,A -85,B 0,C 180,E1 -10956.527,E2 -10956.527} C_VEL
LIN {X 0,Y 408.516,Z 539.098,A -85,B 0,C 180,E1 -10959.694,E2 -10959.694} C_VEL
LIN {X 0,Y 412.087,Z 556.501,A -85,B 0,C 180,E1 -10960.529,E2 -10960.529} C_VEL
LIN {X 0,Y 413.517,Z 566.211,A -85,B 0,C 180,E1 -10960.927,E2 -10960.927} C_VEL
LIN {X 0,Y 410.507,Z 645.809,A -85,B 0,C 180,E1 -10962.951,E2 -10962.951} C_VEL
LIN {X 0,Y 409.923,Z 659.995,A -85,B 0,C 180,E1 -10963.375,E2 -10963.375} C_VEL
LIN {X 0,Y 409.176,Z 674.737,A -85,B 0,C 180,E1 -10964.049,E2 -10964.049} C_VEL
LIN {X 0,Y 408.428,Z 687.137,A -85,B 0,C 180,E1 -10964.831,E2 -10964.831} C_VEL
LIN {X 0,Y 407.673,Z 697.511,A -85,B 0,C 180,E1 -10965.652,E2 -10965.652} C_VEL
LIN {X 0,Y 406.71,Z 708.912,A -85,B 0,C 180,E1 -10966.764,E2 -10966.764} C_VEL
LIN {X 0,Y 405.802,Z 719.215,A -85,B 0,C 180,E1 -10968.005,E2 -10968.005} C_VEL
LIN {X 0,Y 405.189,Z 727.646,A -85,B 0,C 180,E1 -10969.254,E2 -10969.254} C_VEL
LIN {X 0,Y 404.458,Z 735.946,A -85,B 0,C 180,E1 -10970.751,E2 -10970.751} C_VEL
LIN {X 0,Y 403.972,Z 741.601,A -85,B 0,C 180,E1 -10972,E2 -10972} C_VEL
LIN {X 0,Y 403.683,Z 747.115,A -85,B 0,C 180,E1 -10973.502,E2 -10973.502} C_VEL
LIN {X 0,Y 403.201,Z 751.443,A -85,B 0,C 180,E1 -10975,E2 -10975} C_VEL
LIN {X 0,Y 403.256,Z 753.723,A -85,B 0,C 180,E1 -10976.002,E2 -10976.002} C_VEL
LIN {X 0,Y 403.132,Z 755.507,A -85,B 0,C 180,E1 -10977.002,E2 -10977.002} C_VEL
LIN {X 0,Y 402.975,Z 756.854,A -85,B 0,C 180,E1 -10978.001,E2 -10978.001} C_VEL
LIN {X 0,Y 402.888,Z 757.785,A -85,B 0,C 180,E1 -10979,E2 -10979} C_VEL
LIN {X 0,Y 402.852,Z 758.287,A -85,B 0,C 180,E1 -10980,E2 -10980} C_VEL
LIN {X 0,Y 402.867,Z 758.327,A -85,B 0,C 180,E1 -10981,E2 -10981} C_VEL
LIN {X 0,Y 402.921,Z 757.955,A -85,B 0,C 180,E1 -10981.999,E2 -10981.999} C_VEL
LIN {X 0,Y 402.902,Z 757.174,A -85,B 0,C 180,E1 -10983,E2 -10983} C_VEL
LIN {X 0,Y 402.901,Z 755.95,A -85,B 0,C 180,E1 -10984.001,E2 -10984.001} C_VEL
LIN {X 0,Y 403.039,Z 753.278,A -85,B 0,C 180,E1 -10985.503,E2 -10985.503} C_VEL
LIN {X 0,Y 403.114,Z 749.54,A -85,B 0,C 180,E1 -10987.01,E2 -10987.01} C_VEL
LIN {X 0,Y 403.374,Z 744.631,A -85,B 0,C 180,E1 -10988.517,E2 -10988.517} C_VEL
LIN {X 0,Y 403.791,Z 737.235,A -85,B 0,C 180,E1 -10990.277,E2 -10990.277} C_VEL
LIN {X 0,Y 404.324,Z 729.225,A -85,B 0,C 180,E1 -10991.785,E2 -10991.785} C_VEL
LIN {X 0,Y 404.874,Z 719.521,A -85,B 0,C 180,E1 -10993.248,E2 -10993.248} C_VEL
LIN {X 0,Y 405.563,Z 708.822,A -85,B 0,C 180,E1 -10994.553,E2 -10994.553} C_VEL
LIN {X 0,Y 406.372,Z 697.192,A -85,B 0,C 180,E1 -10995.678,E2 -10995.678} C_VEL
LIN {X 0,Y 407.013,Z 685.916,A -85,B 0,C 180,E1 -10996.553,E2 -10996.553} C_VEL
LIN {X 0,Y 407.592,Z 673.561,A -85,B 0,C 180,E1 -10997.304,E2 -10997.304} C_VEL
LIN {X 0,Y 408.125,Z 660.132,A -85,B 0,C 180,E1 -10997.895,E2 -10997.895} C_VEL
LIN {X 0,Y 408.565,Z 646.268,A -85,B 0,C 180,E1 -10998.296,E2 -10998.296} C_VEL
LIN {X 0,Y 410.349,Z 564.847,A -85,B 0,C 180,E1 -11000.073,E2 -11000.073} C_VEL
LIN {X 0,Y 406.608,Z 540.159,A -85,B 0,C 180,E1 -11000.821,E2 -11000.821} C_VEL
LIN {X 0,Y 408.001,Z 520.752,A -85,B 0,C 180,E1 -11004.419,E2 -11004.419} C_VEL
LIN {X 0,Y 409.03,Z 508.164,A -85,B 0,C 180,E1 -11006.782,E2 -11006.782} C_VEL
LIN {X 0,Y 407.397,Z 499.469,A -85,B 0,C 180,E1 -11008.574,E2 -11008.574} C_VEL
LIN {X 0,Y 404.122,Z 485.273,A -85,B 0,C 180,E1 -11011.644,E2 -11011.644} C_VEL
LIN {X 0,Y 404.188,Z 485.262,A -85,B 0,C 180,E1 -11015.016,E2 -11015.016} C_VEL
LIN {X 0,Y 404.162,Z 485.262,A -85,B 0,C 180,E1 -11018.756,E2 -11018.756} C_VEL
LIN {X 0,Y 404.126,Z 485.274,A -85,B 0,C 180,E1 -11021.6,E2 -11021.6} C_VEL
LIN {X 0,Y 404.147,Z 485.263,A -85,B 0,C 180,E1 -11024.522,E2 -11024.522} C_VEL
LIN {X 0,Y 404.138,Z 485.268,A -85,B 0,C 180,E1 -11027.295,E2 -11027.295} C_VEL
LIN {X 0,Y 404.171,Z 485.263,A -85,B 0,C 180,E1 -11029.955,E2 -11029.955} C_VEL
LIN {X 0,Y 404.137,Z 485.267,A -85,B 0,C 180,E1 -11033.125,E2 -11033.125} C_VEL
LIN {X 0,Y 404.147,Z 485.265,A -85,B 0,C 180,E1 -11036.188,E2 -11036.188} C_VEL
LIN {X 0,Y 404.147,Z 485.269,A -85,B 0,C 180,E1 -11039.715,E2 -11039.715} C_VEL
LIN {X 0,Y 404.197,Z 485.26,A -85,B 0,C 180,E1 -11043.123,E2 -11043.123} C_VEL
LIN {X 0,Y 404.179,Z 485.264,A -85,B 0,C 180,E1 -11045.334,E2 -11045.334} C_VEL
LIN {X 0,Y 404.141,Z 485.264,A -85,B 0,C 180,E1 -11048.581,E2 -11048.581} C_VEL
LIN {X 0,Y 404.212,Z 485.26,A -85,B 0,C 180,E1 -11051.762,E2 -11051.762} C_VEL
LIN {X 0,Y 404.209,Z 485.257,A -85,B 0,C 180,E1 -11054.882,E2 -11054.882} C_VEL
LIN {X 0,Y 404.258,Z 485.252,A -85,B 0,C 180,E1 -11057.958,E2 -11057.958} C_VEL
LIN {X 0,Y 404.435,Z 485.229,A -85,B 0,C 180,E1 -11062.1,E2 -11062.1} C_VEL
LIN {X 0,Y 404.426,Z 485.23,A -85,B 0,C 180,E1 -11064.015,E2 -11064.015} C_VEL
LIN {X 0,Y 404.484,Z 485.223,A -85,B 0,C 180,E1 -11068.008,E2 -11068.008} C_VEL
LIN {X 0,Y 404.613,Z 485.207,A -85,B 0,C 180,E1 -11070,E2 -11070} C_VEL
LIN {X 0,Y 404.425,Z 485.231,A -85,B 0,C 180,E1 -11072.961,E2 -11072.961} C_VEL
